# B&R Automation Studio project Parker_BMM_ST_V5_3147_V12 (part 26)

#### extruder.c - Implementation code
```c
/********************************************************************
 * COPYRIGHT --
 ********************************************************************
 * Program: extruder
 * File: extruder.c
 * Author: lij
 * Created: January 05, 2015
 ********************************************************************
 * Implementation of program extruder
 ********************************************************************/

#include <bur/plctypes.h>

#ifdef _DEFAULT_INCLUDES
	#include <AsDefault.h>
#endif

/**************************************************************************************
** 					               include user files								 **
**************************************************************************************/
#include "edge.h"               /*edge function                         */
#include "keyap2100.h"
//#include "keyap880.h"
#include "pic_id.h"

/**************************************************************************************
** 					 	                 define								                   **
**************************************************************************************/
#define     S$EXTRUDER_WAIT		           	 0
#define     S$EXTRUDER_CONTACTOR_ON		   	10
#define     S$EXTRUDER_POWER_ON_DELAY			20
#define     S$EXTRUDER_POWER_ON		        	30
#define     S$EXTRUDER_READY		       		100
#define     S$EXTRUDER_BASIC_ZONE		  		110
#define     S$EXTRUDER_PRODUCTION_ZONE	   	130
#define     S$EXTRUDER_DEC_ZONE		       	150
#define     S$EXTRUDER_POWER_OFF_DECEL			200
#define     S$EXTRUDER_POWER_OFF_PROTECT		210
#define     S$EXTRUDER_POWER_OFF_DELAY			220
/**************************************************************************************
                               Function Declarations
**************************************************************************************/
void SpeedUpDw(short ins_des,short command,speedAdjust_typ * pSpeedUpDwData);

void ExtruderCtrl(Extruder_Ctrl_typ * pExtruder,Extruder_Para_typ * pExtrPara,speedAdjust_typ * pSpeedUpDwData, Lubricate_Check_typ * pLubricCheck);

/**************************************************************************************
     	        	       I N I T U P  O F   T H E   T A S K
**************************************************************************************/
void _INIT extruderINIT(void)
{
	/* TODO: Add code here */
    RTInfo_Task.enable = 1;
    RTInfo(&RTInfo_Task);

    tTask = RTInfo_Task.cycle_time/1000.0/1000.0;		/*  from us ---> s  */

    MotorSpeedA.minVal  	  = 0;
    MotorSpeedA.frequence	  = 30;
    MotorSpeedA.waitTimeSlow = 200;
    MotorSpeedA.waitTimeFast = 500;
    MotorSpeedA.unitsSlow    = 1;
    MotorSpeedA.unitsFast	= 5;
    MotorSpeedA.unitsVFast	= 20;

    MotorSpeedA.maxVal = 100;
    MotorSpeedA.minVal = 0;

    MotorSpeedB.minVal  	 = 0;
    MotorSpeedB.frequence	 = 30;
    MotorSpeedB.waitTimeSlow = 200;
    MotorSpeedB.waitTimeFast = 500;
    MotorSpeedB.unitsSlow    = 1;
    MotorSpeedB.unitsFast	 = 5;
    MotorSpeedB.unitsVFast	 = 20;

    MotorSpeedB.maxVal = 100;
    MotorSpeedB.minVal = 0;

    MotorSpeedVisu.frequence	= 30;
    MotorSpeedVisu.waitTimeSlow = 200;
    MotorSpeedVisu.waitTimeFast = 500;
    MotorSpeedVisu.unitsSlow    = 1;
    MotorSpeedVisu.unitsFast	= 5;
    MotorSpeedVisu.unitsVFast	= 20;

    MotorSpeedVisu.maxVal = 100;
    MotorSpeedVisu.minVal = 0;

    cntExtruderStopDelay = 0;

    gExtruderA.Step = S$EXTRUDER_WAIT;
    gExtruderB.Step = S$EXTRUDER_WAIT;
    gExtruderVisu.Step = S$EXTRUDER_WAIT;

    gExtruderA.tTask  = tTask;
    gExtruderB.tTask  = tTask;
    gExtruderVisu.tTask = tTask;

	bHideCurrencyA = 0;
	bHideMeltTempA = 1;
	bHidePressureA = 1;

	bHideCurrencyB = 0;
	bHideMeltTempB = 1;
	bHidePressureB = 1;

	bHideCurrencyV = 1;
	bHideMeltTempV = 1;
	bHidePressureV = 1;

}
/**************************************************************************************
        				   C Y C L I C   P A R T   O F   T H E   T A S K
**************************************************************************************/
void _CYCLIC extruderCYCLIC(void)
{
	if(0 == gMachineFix.ExtruderA.RPM10v )gMachineFix.ExtruderA.RPM10v = 1500;
	if(0 == gMachineFix.ExtruderB.RPM10v)gMachineFix.ExtruderB.RPM10v  = 1500;
	if(0 == gMachineFix.ExtruderVisu.RPM10v )gMachineFix.ExtruderVisu.RPM10v = 1500;

	if(0 == gMachineFix.ExtruderA.Currency10V )gMachineFix.ExtruderA.Currency10V = 50;
	if(0 == gMachineFix.ExtruderB.Currency10V)gMachineFix.ExtruderB.Currency10V= 50;
	if(0 == gMachineFix.ExtruderVisu.Currency10V )gMachineFix.ExtruderVisu.Currency10V = 50;

	/*  -------------------- Extruder motor speed and current -------------------------- */
	if(gMachineOut.ExtrA_On)
	{
		gExtruderA.MotorRPM = gExtruderA.aiActRPM/32767.0  * gMachineFix.ExtruderA.RPM10v;
		gExtruderA.Current  = gExtruderA.aiCurrent/32767.0 * gMachineFix.ExtruderA.Currency10V;
		gExtruderA.ActRPM   = gExtruderA.ActSpeed/100.0  * gMachineFix.ExtruderA.RPM10v;
	}
	else
	{
		gExtruderA.MotorRPM = 0.0;
		gExtruderA.Current  = 0.0;
		gExtruderA.ActRPM   = 0.0;
	}

	if(gMachineOut.ExtrB_On)
	{
		gExtruderB.MotorRPM = gExtruderB.aiActRPM/32767.0  * gMachineFix.ExtruderB.RPM10v;
		gExtruderB.Current  = gExtruderB.aiCurrent/32767.0 * gMachineFix.ExtruderB.Currency10V;
	}
	else
	{
		gExtruderB.MotorRPM = 0.0;
		gExtruderB.Current  = 0.0;
	}

	if(gMachineOut.ExtrVisu_On)
	{
		gExtruderVisu.MotorRPM = gExtruderVisu.aiActRPM/32767.0  * gMachineFix.ExtruderVisu.RPM10v;
		gExtruderVisu.Current  = gExtruderVisu.aiCurrent/32767.0 * gMachineFix.ExtruderVisu.Currency10V;
	}
	else
	{
		gExtruderVisu.MotorRPM = 0.0;
		gExtruderVisu.Current  = 0.0;
	}

	/* ------------------ Extruder zero and max pressure ------------------ */
	if((1 == btnZeroExtrA) && (0 == btnZeroExtrA_POS))
	{
		gMachineFix.ExtruderA.MeltP0V = gExtruderA.aiMeltPressure/3276.7;
		gRecipeOperate.OnceSave = 1;
	}

	if(1 == btnMaxExtrA)
	{
		gMachineOut.MeltPrShunt = 1;
		tMaxExtrA = tMaxExtrA + tTask;
	}
	else
	{
		tMaxExtrA = 0.0;
	}

	if(tMaxExtrA > 3.0 - tTask  && tMaxExtrA < 3.0 + tTask  )
	{
		gMachineFix.ExtruderA.MeltP10V = gExtruderA.aiMeltPressure/3276.7;
		gRecipeOperate.OnceSave = 1;
	}

	if((1 == btnZeroExtrB) && (0 == btnZeroExtrB_POS))
	{
		gMachineFix.ExtruderB.MeltP0V = gHardWare.AI4632_3[1]/3276.7;		/* no this input  */
		gRecipeOperate.OnceSave = 1;
	}

	if(1 == btnMaxExtrB)
	{
		gMachineOut.MeltPrShunt = 1;
		tMaxExtrB = tMaxExtrB + tTask;
	}
	else
	{
		tMaxExtrB = 0.0;
	}

	if(tMaxExtrB > 3.0 - tTask  && tMaxExtrB < 3.0 + tTask )
	{
		gMachineFix.ExtruderB.MeltP10V = gHardWare.AI4632_3[1]/3276.7;
		gRecipeOperate.OnceSave = 1;
	}

	if(0 == btnMaxExtrA && 0 == btnMaxExtrB)
	{
		gMachineOut.MeltPrShunt = 0;
	}
	/*  -------------------- Melt pressure alarm  -------------------------- */
	if(gMachineFix.ExtruderA.WarningMeltP < 50)gMachineFix.ExtruderA.WarningMeltP = 50.0;
	if(gMachineFix.ExtruderA.AlarmMeltP < 100)gMachineFix.ExtruderA.AlarmMeltP = 100.0;

	if(gExtruderA.aiMeltPressure != 32767)
	{
		if(gExtruderA.MeltPressure > gMachineFix.ExtruderA.AlarmMeltP)
		{
			if(0 == btnMaxExtrA)
			{
				gAlarm.ExtrAMeltP_Alarm = 1;
				gAlarm.ExtrAMeltP_Warn  = 0;
			}
		}
		else if(gExtruderA.MeltPressure > gMachineFix.ExtruderA.WarningMeltP)
		{
			gAlarm.ExtrAMeltP_Alarm = 0;
			gAlarm.ExtrAMeltP_Warn  = 1;
		}
		else
		{
			gAlarm.ExtrAMeltP_Alarm = 0;
			gAlarm.ExtrAMeltP_Warn  = 0;
		}
	}
	else
	{
		gAlarm.ExtrAMeltP_Alarm = 0;
		gAlarm.ExtrAMeltP_Warn  = 0;
	}

	/* --------------------  current alarm and warning -------------------- */
	if(gMachineFix.ExtruderA.WarningCurrent < 2)gMachineFix.ExtruderA.WarningCurrent = 2;
	if(gMachineFix.ExtruderA.AlarmCurrent   < 5)gMachineFix.ExtruderA.AlarmCurrent = 5;

	if(gExtruderA.aiCurrent != 32767)
	{
		if(gExtruderA.Current > gMachineFix.ExtruderA.AlarmCurrent)
		{
			tAlarmCurentA = tAlarmCurentA+tTask;
			if(tAlarmCurentA > 10000)tAlarmCurentA= 1000;
			tWarnCurentA  = 0.0;
		}
		else if(gExtruderA.Current > gMachineFix.ExtruderA.WarningCurrent)
		{
			tAlarmCurentA = 0.0;
			tWarnCurentA = tWarnCurentA+tTask;
			if(tWarnCurentA > 10000)tWarnCurentA = 1000;
		}
		else
		{
			tWarnCurentA = 0.0;
			tAlarmCurentA = 0.0;
		}

		if(tAlarmCurentA > 5.0)
		{
			gAlarm.ExtrACurrentAlarm = 1;
		}
		else
		{
			gAlarm.ExtrACurrentAlarm = 0;
		}

		if(tWarnCurentA > 5.0)
		{
			gAlarm.ExtrACurrentWarn = 1;
		}
		else
		{
			gAlarm.ExtrACurrentWarn = 0;
		}
	}
	else
	{
		tWarnCurentA = 0.0;
		tAlarmCurentA = 0.0;

		gAlarm.ExtrACurrentWarn = 0;
		gAlarm.ExtrACurrentAlarm = 0;
	}

	if(gMachineFix.ExtruderB.WarningCurrent < 2)gMachineFix.ExtruderB.WarningCurrent = 2;
	if(gMachineFix.ExtruderB.AlarmCurrent   < 5)gMachineFix.ExtruderB.AlarmCurrent = 5;

	if(gExtruderB.aiCurrent != 32767)
	{
		if(gExtruderB.Current > gMachineFix.ExtruderB.AlarmCurrent)
		{
			tAlarmCurentB = tAlarmCurentB+tTask;
			if(tAlarmCurentB > 10000)tAlarmCurentB= 1000;
			tWarnCurentB  = 0.0;
		}
		else if(gExtruderB.Current > gMachineFix.ExtruderB.WarningCurrent)
		{
			tAlarmCurentB = 0.0;
			tWarnCurentB = tWarnCurentB+tTask;
			if(tWarnCurentB > 10000)tWarnCurentB = 1000;
		}
		else
		{
			tWarnCurentB = 0.0;
			tAlarmCurentB = 0.0;
		}

		if(tAlarmCurentB > 5.0)
		{
			gAlarm.ExtrBCurrentAlarm = 1;
		}
		else
		{
			gAlarm.ExtrBCurrentAlarm = 0;
		}

		if(tWarnCurentB > 5.0)
		{
			gAlarm.ExtrBCurrentWarn = 1;
		}
		else
		{
			gAlarm.ExtrBCurrentWarn = 0;
		}
	}
	else
	{
		tWarnCurentB = 0.0;
		tAlarmCurentB = 0.0;

		gAlarm.ExtrBCurrentWarn = 0;
		gAlarm.ExtrBCurrentAlarm = 0;
	}

	/* -------------------- Hopper cooling  -------------------------- */
	bHideHopperCooling = !gMachineFix.Option.bHopperCooling;
	gMachineFix.Option.bHopperCooling =0; //ipis0319
	if(1 == gMachineFix.Option.bHopperCooling)
	{
		if(!gMachinePara.HopperCoolStart)gMachinePara.HopperCoolStart = 65;
		if(!gMachinePara.HopperCoolStop )gMachinePara.HopperCoolStop = 55;

		if(gMachineInfo.TempHopper > gMachinePara.HopperCoolStart)
		{
			gMachineOut.HopperCoolingA = 1;
		}

		if(gMachineInfo.TempHopper < gMachinePara.HopperCoolStop)
		{
			gMachineOut.HopperCoolingA = 0;
		}
	}
	else
	{
		gMachineOut.HopperCoolingA = 0;
	}
	/* -------------------- Extruder motor cooling  -------------------------- */
	bHideExtrMotorCooling = !gMachineFix.Option.bExtruderMotorCooling;
	gMachineFix.Option.bExtruderMotorCooling=0; //ipis0319
	if(!gMachinePara.ExtruderA.TempCoolStart)gMachinePara.ExtruderA.TempCoolStart = 75;
	if(!gMachinePara.ExtruderA.TempCoolStop)gMachinePara.ExtruderA.TempCoolStop = 65;
	if(!gMachinePara.ExtrLiftLower.warningMotorTemp)gMachinePara.ExtrLiftLower.warningMotorTemp= 90;
	if(!gMachinePara.ExtrLiftLower.AlarmMotorTemp)gMachinePara.ExtrLiftLower.AlarmMotorTemp = 100;

	if(1 == gMachineFix.Option.bExtruderMotorCooling)
	{
		if(gMachineInfo.TempExtrCoolWater > gMachinePara.ExtruderA.TempCoolStart)
		{
			gMachineOut.ExtrA_CoolWaterOn = 1;
		}

		if(gMachineInfo.TempExtrCoolWater < gMachinePara.ExtruderA.TempCoolStop)
		{
			gMachineOut.ExtrA_CoolWaterOn = 0;
		}

		if(gMachineInfo.TempExtrCoolWater > gMachinePara.ExtrLiftLower.warningMotorTemp)
		{
			tAlarmExtrTempA = tAlarmExtrTempA + tTask;

			if(tAlarmExtrTempA > 10000.0)tAlarmExtrTempA = 100.0;
		}
		else
		{
			tAlarmExtrTempA = 0.0;
		}

		if(tAlarmExtrTempA > 10.0)
		{
			gAlarm.A_ExtrMotorTempAlarm = 1;
		}

		if(gMachineInfo.TempExtrCoolWater > gMachinePara.ExtrLiftLower.AlarmMotorTemp)
		{
			tStopExtrTempA = tStopExtrTempA + tTask;

			if(tStopExtrTempA > 10000.0)tStopExtrTempA = 100.0;
		}
		else
		{
			tStopExtrTempA = 0.0;
		}

		if(tStopExtrTempA > 10.0)
		{
			gAlarm.A_ExtrMotorTempStop = 1;
		}

		if(0 == gMachineIn.ExtrA_ColiTempNormal)
		{
			tColiTempNormalA = tColiTempNormalA + tTask;

			if(tColiTempNormalA > 10000.0)tColiTempNormalA = 100.0;
		}
		else
		{
			tColiTempNormalA = 0.0;
		}

		if(tColiTempNormalA > 10.0)
		{
			gAlarm.A_ColiTempNormal = 1;
		}
	}
	else
	{
		gAlarm.A_ExtrMotorTempStop = 0;
		gAlarm.A_ColiTempNormal = 0;
		gMachineOut.ExtrA_CoolWaterOn = 0;
	}

   /* ----------------------- extruder key ------------------------- */
   if(1 == gMachineIn.MainControl && gPanelObj.GetPicture != PIC_INIT && gPanelObj.GetPicture != PIC_SCREEN_SAVE)
   {
     gExtruderA.bKeyOnOff       = gPanelObj.KeyMatric[S$KEYMATRIX_EXTRUDER_A];
     gExtruderB.bKeyOnOff    = gPanelObj.KeyMatric[S$KEYMATRIX_EXTRUDER_B];
	  gMachineIn.ExtrA_HopperKey = gPanelObj.KeyMatric[S$KEYMATRIX_HOPPER_A];
   }/*if(1 == gMachineIn.MainControl ..... */

   /* ----- A extruder increase or decrease speed ----- */
   if(16384 == gExtruderA.FoucsBasic || 16384 == gExtruderA.FocusProduct || PIC_SPEED != gPanelObj.GetPicture)
   {
      gExtruderA.bKeyInc = gPanelObj.KeyMatric[S$KEYMATRIX_SPEED_UP];
      gExtruderA.bKeyDec = gPanelObj.KeyMatric[S$KEYMATRIX_SPEED_DN];
   }
   else
   {
      gExtruderA.bKeyInc = 0;
      gExtruderA.bKeyDec = 0;
   }
   gExtruderA.tProtect = gMachineFix.ExtruderA.tProtect;
   gExtruderA.tOnDelay = gMachineFix.ExtruderA.tOnDelay;
   gExtruderA.tOffDelay = gMachineFix.ExtruderA.tOffDelay;

	LubricCheckA.diLubricCheck = gMachineIn.ExtrA_LubrNormal;
	LubricCheckA.tSetCheckTime = gMachineFix.ExtruderA.tLubricateCheck;

   ExtruderCtrl(&gExtruderA, &gMachinePara.ExtruderA, &MotorSpeedA, &LubricCheckA);
   gMachineOut.ExtrA_On = gExtruderA.doOn;

	gAlarm.A_ExtrLubricCheck = LubricCheckA.bLubricError;
//	gAlarm.A_ExtruderMotorOverload = gMachineIn.ExtrA_MotorErr;

	/* extruder A on and feedback  */
	gMachineIn.ExtrA_OnOff = gMachineOut.ExtrA_On;
	if(gMachineOut.ExtrA_On != gMachineIn.ExtrA_OnOff)
	{
		tExtrA_OnNormal = tExtrA_OnNormal + tTask;
		if(tExtrA_OnNormal >= 600.0)tExtrA_OnNormal = 60.0;
	}
	else
	{
		tExtrA_OnNormal = 0.0;
	}

	if(tExtrA_OnNormal >= 30.0)
	{
		gExtruderA.OnFeedbackErr = 1;
		gAlarm.ExtrA_NotOn = 1;
	}
	else
	{
		gExtruderA.OnFeedbackErr = 0;
	}

	/*  extruder A hopper  */
	if(1 == gMachineIn.ExtrA_HopperKey && 0 == ExtrA_HopperKeyOld)
	{
		if((1 == gMachineIn.ExtrA_OnOff) && (gExtruderA.Out > 0.0))
		{
			gMachineOut.HopperGateOpenA = !gMachineOut.HopperGateOpenA;
		}
		else
		{
			if(0 == gMachineIn.ExtrA_OnOff)gImply.ExtruderA_NotOn = 1;
			if(0.0 == gExtruderA.Out)gImply.ExtruderA_NotOut = 1;
		}
	}
	ExtrA_HopperKeyOld = gMachineIn.ExtrA_HopperKey;

	if((0 == gMachineIn.ExtrA_OnOff) || (0.0 == gExtruderA.Out))
	{
		if(1 == gMachineOut.HopperGateOpenA)
		{
			if(0 == gMachineIn.ExtrA_OnOff)gImply.ExtruderA_NotOn = 1;
			if(0.0 == gExtruderA.Out)gImply.ExtruderA_NotOut = 1;
			gMachineOut.HopperGateOpenA = 0;
		}
	}

   /* ----- B extruder increase or decrease speed ----- */
   if(16384 == gExtruderB.FoucsBasic || 16384 == gExtruderB.FocusProduct)
   {
      gExtruderB.bKeyInc = gPanelObj.KeyMatric[S$KEYMATRIX_SPEED_UP];
      gExtruderB.bKeyDec = gPanelObj.KeyMatric[S$KEYMATRIX_SPEED_DN];
   }
   else
   {
      gExtruderB.bKeyInc = 0;
      gExtruderB.bKeyDec = 0;
   }
   gExtruderB.tProtect = gMachineFix.ExtruderA.tProtect;
   gExtruderB.tOnDelay = gMachineFix.ExtruderA.tOnDelay;
   gExtruderB.tOffDelay = gMachineFix.ExtruderA.tOffDelay;

	LubricCheckB.diLubricCheck = gMachineIn.ExtrB_LubrNormal;
	LubricCheckB.tSetCheckTime = gMachineFix.ExtruderA.tLubricateCheck;

   ExtruderCtrl(&gExtruderB, &gMachinePara.ExtruderB, &MotorSpeedB, &LubricCheckB);
   gMachineOut.ExtrB_On = gExtruderB.doOn;

	gAlarm.B_ExtrLubricCheck = LubricCheckB.bLubricError;
//	gAlarm.B_ExtruderMotorOverload = gMachineIn.ExtrB_MotorErr;

	/* extruder B on and feedback  */
	gMachineIn.ExtrB_OnOff = gMachineOut.ExtrB_On;
	if(gMachineOut.ExtrB_On != gMachineIn.ExtrB_OnOff)
	{
		tExtrB_OnNormal = tExtrA_OnNormal + tTask;
		if(tExtrB_OnNormal >= 600.0)tExtrB_OnNormal = 60.0;
	}
	else
	{
		tExtrB_OnNormal = 0.0;
	}

	if(tExtrB_OnNormal >= 30.0)
	{
		gExtruderB.OnFeedbackErr = 1;
		gAlarm.ExtrB_NotOn = 1;
	}
	else
	{
		gExtruderB.OnFeedbackErr = 0;
	}

	if(1 == gMachineIn.ExtrB_HopperKey && 0 == ExtrB_HopperKeyOld)
	{
		if((1 == gMachineIn.ExtrB_OnOff) && (gExtruderB.Out > 0.0))
		{
			gMachineOut.HopperGateOpenB = !gMachineOut.HopperGateOpenB;
		}
		else
		{
			if(0 == gMachineIn.ExtrB_OnOff)gImply.ExtruderB_NotOn = 1;
			if(0.0 == gExtruderB.Out)gImply.ExtruderB_NotOut = 1;
		}
	}
	ExtrB_HopperKeyOld = gMachineIn.ExtrB_HopperKey;

	if((0 == gMachineIn.ExtrB_OnOff) || (0.0 == gExtruderB.Out))
	{
		if(1 == gMachineOut.HopperGateOpenB)
		{
			if(0 == gMachineIn.ExtrB_OnOff)gImply.ExtruderB_NotOn = 1;
			if(0.0 == gExtruderB.Out)gImply.ExtruderB_NotOut = 1;
			gMachineOut.HopperGateOpenB = 0;
		}
	}

   /* ----- Visual extruder increase or decrease speed ----- */
   if(16384 == gExtruderVisu.FoucsBasic || 16384 == gExtruderVisu.FocusProduct)
   {
      gExtruderVisu.bKeyInc = gPanelObj.KeyMatric[S$KEYMATRIX_SPEED_UP];
      gExtruderVisu.bKeyDec = gPanelObj.KeyMatric[S$KEYMATRIX_SPEED_DN];
   }
   else
   {
      gExtruderVisu.bKeyInc = 0;
      gExtruderVisu.bKeyDec = 0;
   }
   gExtruderVisu.tProtect = gMachineFix.ExtruderA.tProtect;
   gExtruderVisu.tOnDelay = gMachineFix.ExtruderA.tOnDelay;
   gExtruderVisu.tOffDelay = gMachineFix.ExtruderA.tOffDelay;

	LubricCheckVisu.diLubricCheck = 1;
	LubricCheckVisu.tSetCheckTime = gMachineFix.ExtruderA.tLubricateCheck;

   ExtruderCtrl(&gExtruderVisu, &gMachinePara.ExtruderVisu, &MotorSpeedVisu, &LubricCheckVisu);
   gMachineOut.ExtrVisu_On = gExtruderVisu.doOn;

	gAlarm.VisuExtrMotorOverload = gMachineIn.ExtrV_MotorErr;
	gAlarm.VisuExtrCoolOverload  = gMachineIn.ExtrV_CoolMotorErr;

	/* extruder A on and feedback  */
	if(gMachineOut.ExtrVisu_On != gMachineIn.ExtrV_OnOff)
	{
		tExtrV_OnNormal = tExtrV_OnNormal + tTask;
		if(tExtrV_OnNormal >= 600.0)tExtrV_OnNormal = 60.0;
	}
	else
	{
		tExtrV_OnNormal = 0.0;
	}

	if(tExtrV_OnNormal >= 30.0)
	{
		gExtruderVisu.OnFeedbackErr = 1;
		gAlarm.ExtrV_NotOn = 1;
	}
	else
	{
		gExtruderVisu.OnFeedbackErr = 0;
	}

   gMachineInfo.Extruder       = gMachineOut.ExtrA_On;
   gMachineOut.ExtruderCooling = gMachineInfo.Extruder;

   /* ----------------------- Stop extruder ----------------------- */
   /* ----- A extruder ----- */
   gExtruderA.bKeyOff = 0;
   if (1 == gMachineInfo.ExtrTLow     || 0 == gMachineInfo.IsHeat           || 0 == gMachineIn.ParisonPumpRunning   ||
       1 == gMachineIn.ExtrA_MotorErr || 1 == gMachineIn.ExtrA_CoolMotorErr || 1 == gAlarm.A_ExtrMotorTempStop      ||
		 1 == gAlarm.ExtrACurrentAlarm)
   {
		if(1 == gMachineOut.ExtrA_On)
		{
			if(1 == gMachineInfo.ExtrTLow)gAlarm.ScrewTempLow = 1;
			if(0 == gMachineInfo.IsHeat)gAlarm.HeatingNotOn = 1;
			if(0 == gMachineIn.ParisonPumpRunning)gAlarm.ParisonPumpNotOn = 1;
//			gAlarm.A_ExtruderMotorOverload = gMachineIn.ExtrA_MotorErr;
			gExtruderA.bKeyOff = 1;
		}
   }

   /* ----- B extruder ----- */
   gExtruderB.bKeyOff = 0;
   if (1 == gMachineInfo.ExtrTLow     || 0 == gMachineInfo.IsHeat           || 0 == gMachineIn.ParisonPumpRunning ||
       1 == gMachineIn.ExtrB_MotorErr || 1 == gMachineIn.ExtrB_CoolMotorErr || 1 == gAlarm.ExtrBCurrentAlarm)
   {
		if(1 == gMachineOut.ExtrB_On)
		{
			if(1 == gMachineInfo.ExtrTLow)gAlarm.ScrewTempLow = 1;
			if(0 == gMachineInfo.IsHeat)gAlarm.HeatingNotOn = 1;
			if(0 == gMachineIn.ParisonPumpRunning)gAlarm.ParisonPumpNotOn = 1;
//			gAlarm.B_ExtruderMotorOverload = gMachineIn.ExtrB_MotorErr;
			gExtruderB.bKeyOff = 1;
		}
   }

   /* ----- Visual extruder ----- */
   gExtruderVisu.bKeyOff = 0;
   if (1 == gMachineInfo.ExtrTLow     || 0 == gMachineInfo.IsHeat || 0 == gMachineIn.ParisonPumpRunning ||
       1 == gMachineIn.ExtrV_MotorErr || 1 == gMachineIn.ExtrV_CoolMotorErr || 0 == gMachineIn.ExtrA_OnOff)
   {
		if(1 == gMachineOut.ExtrVisu_On)
		{
			if(1 == gMachineInfo.ExtrTLow)gAlarm.ScrewTempLow = 1;
			if(0 == gMachineInfo.IsHeat)gAlarm.HeatingNotOn = 1;
			if(0 == gMachineIn.ParisonPumpRunning)gAlarm.ParisonPumpNotOn = 1;
			gAlarm.VisuExtrMotorOverload = gMachineIn.ExtrV_MotorErr;
			if(0 == gMachineIn.ExtrA_OnOff)gAlarm.ExtrA_NotOn = 1;
			gExtruderVisu.bKeyOff = 1;
		}
   }

   /* ------------------------ Auto error stop extruder ---------------------------- */
   if(1 == gPROCESS_info.extruderStopEnable)
   {
     cntExtruderStopDelay ++;
   }
   else
   {
     cntExtruderStopDelay = 0;
   }

   if(gMachineFix.ExtruderA.StopTime <= 0.0)gMachineFix.ExtruderA.StopTime = 3.0;
   if(gMachineFix.ExtruderA.StopTime < cntExtruderStopDelay * tTask)
   {
     if(1 == gTKmanual.Status)
     {
         gExtruderA.bKeyOff = 1;
         gExtruderB.bKeyOff = 1;
		 gExtruderD.bKeyOff = 1;
         gExtruderVisu.bKeyOff = 1;
         gPROCESS_info.extruderStopEnable = 0;
         cntExtruderStopDelay = 0;
     }
   }
}
/**************************************************************************************
        				   E X I T   P A R T   O F   T H E   T A S K
**************************************************************************************/
void _EXIT extruderEXIT(void)
{
	/* TODO: Add code here */
}

/* adjust the speed of motor*/
void SpeedUpDw(short ins_des,short command,speedAdjust_typ * pSpeedUpDwData)
{
    unsigned short index;

    if(pSpeedUpDwData->pSpeed != 0)  /*  point is not NULL  */
    {
        index = ins_des + 1;

        if (command == 1)
        {
            pSpeedUpDwData->iSpeed[index]++;
            pSpeedUpDwData->iSpeed[index+1]++;
            if (pSpeedUpDwData->iSpeed[index+1] == 1) (*pSpeedUpDwData->pSpeed) = (*pSpeedUpDwData->pSpeed) + pSpeedUpDwData->unitsSlow*ins_des;
            if (pSpeedUpDwData->iSpeed[index]>pSpeedUpDwData->frequence) pSpeedUpDwData->iSpeed[index] = 0;

            if (pSpeedUpDwData->iSpeed[index+1]<50) ;
            else if (pSpeedUpDwData->iSpeed[index+1]<pSpeedUpDwData->waitTimeSlow)
            {
                if (pSpeedUpDwData->iSpeed[index]== 0) (*pSpeedUpDwData->pSpeed) = (*pSpeedUpDwData->pSpeed) + pSpeedUpDwData->unitsSlow*ins_des;
            }
            else if (pSpeedUpDwData->iSpeed[index+1]<pSpeedUpDwData->waitTimeFast)
            {
                if (pSpeedUpDwData->iSpeed[index] == 0) (*pSpeedUpDwData->pSpeed) = (*pSpeedUpDwData->pSpeed) + pSpeedUpDwData->unitsFast*ins_des;
            }
            else
            {
                if (pSpeedUpDwData->iSpeed[index] == 0) (*pSpeedUpDwData->pSpeed) = (*pSpeedUpDwData->pSpeed) + pSpeedUpDwData->unitsVFast*ins_des;
                pSpeedUpDwData->iSpeed[index+1] = pSpeedUpDwData->waitTimeFast;
            }
        }
        else
        {
            pSpeedUpDwData->iSpeed[index] = 0;
            pSpeedUpDwData->iSpeed[index+1] = 0;
        }
        if ((*pSpeedUpDwData->pSpeed) >= pSpeedUpDwData->maxVal) (*pSpeedUpDwData->pSpeed) = pSpeedUpDwData->maxVal;
        if ((*pSpeedUpDwData->pSpeed) <= pSpeedUpDwData->minVal) (*pSpeedUpDwData->pSpeed) = pSpeedUpDwData->minVal;
    }/*  if(pSpeedUpDwData->pSpeed != 0) */
}/*end of function*/

/* ---------- Extruder contorl ---------- */
void ExtruderCtrl(Extruder_Ctrl_typ * pExtruder, Extruder_Para_typ * pExtrPara, speedAdjust_typ * pSpeedUpDwData, Lubricate_Check_typ * pLubricCheck)
{
    if(pExtruder->tOnDelay  < pExtruder->tTask * 2.0)pExtruder->tOnDelay = pExtruder->tTask * 2.0;
    if(pExtruder->tOffDelay < pExtruder->tTask * 2.0)pExtruder->tOffDelay= pExtruder->tTask * 2.0;

    if(pExtruder->tTask <= 0.0)
    {
        pExtruder->tET_s = 0.0;
        pExtruder->LedOn = 0;
        pExtruder->LedProduction = 0;

        pExtruder->doContactor = 0;
        pExtruder->doOn = 0;
        pExtruder->Out = 0.0;

        pExtruder->bKeyOnOff = 0;
        pExtruder->bKeyOff = 0;
        pExtruder->bKeyOnOffOld = 0;
        pExtruder->bKeyOffOld = 0;

        pExtruder->Step = S$EXTRUDER_WAIT;
        return;
    }

    /*  On Off button edge start */
    if(1 == pExtruder->bKeyOnOff && 0 == pExtruder->bKeyOnOffOld)
    {
        if(S$EXTRUDER_WAIT == pExtruder->Step)
        {
				pExtruder->LedOn = 1;
            pExtruder->Step = S$EXTRUDER_CONTACTOR_ON;
        }
        else
        {
				pExtruder->LedOn = 0;
            if(pExtruder->Step < S$EXTRUDER_POWER_ON && pExtruder->Step > S$EXTRUDER_WAIT)
            {
               pExtruder->Step = S$EXTRUDER_WAIT;
            }
            else if(pExtruder->Step >= S$EXTRUDER_POWER_ON && pExtruder->Step < S$EXTRUDER_POWER_OFF_DECEL)
            {
                if(pExtruder->Step > S$EXTRUDER_BASIC_ZONE)
                {
                    pExtruder->Step = S$EXTRUDER_POWER_OFF_DECEL;
                }
                else
                {
                    pExtruder->Step = S$EXTRUDER_POWER_OFF_PROTECT;
                }
            }
        }
    }
    pExtruder->bKeyOnOffOld = pExtruder->bKeyOnOff;

    /* -------- internal stop -------- */
    if(1 == pExtruder->bKeyOff)
    {
		 pExtruder->LedOn = 0;
       if(pExtruder->Step < S$EXTRUDER_POWER_ON && pExtruder->Step > S$EXTRUDER_WAIT)
       {
          pExtruder->Step = S$EXTRUDER_WAIT;
       }
       else if(pExtruder->Step >= S$EXTRUDER_POWER_ON && pExtruder->Step < S$EXTRUDER_POWER_OFF_DECEL)
       {
          if(pExtruder->Step > S$EXTRUDER_BASIC_ZONE)
          {
             pExtruder->Step = S$EXTRUDER_POWER_OFF_DECEL;
          }
          else
          {
             pExtruder->Step = S$EXTRUDER_POWER_OFF_PROTECT;
          }
       }
    }
    pExtruder->bKeyOffOld = pExtruder->bKeyOff;

	if(1 == pExtruder->bKeyStop)
	{
		pExtruder->bKeyStop = 0;
		if(pExtruder->Step < S$EXTRUDER_POWER_ON && pExtruder->Step > S$EXTRUDER_WAIT)
		{
			pExtruder->Step = S$EXTRUDER_WAIT;
		}
		else if(pExtruder->Step >= S$EXTRUDER_POWER_ON && pExtruder->Step < S$EXTRUDER_POWER_OFF_DECEL)
		{
			if(pExtruder->Step > S$EXTRUDER_BASIC_ZONE)
			{
				pExtruder->Step = S$EXTRUDER_POWER_OFF_DECEL;
			}
			else
			{
				pExtruder->Step = S$EXTRUDER_POWER_OFF_PROTECT;
			}
		}
	}

    /*  ------ motor protection ------- */
    if(pExtruder->doOnOld != pExtruder->doOn && pExtruder->tTask > 0.0)
    {
        pExtruder->cntProtect = pExtruder->tProtect /pExtruder->tTask;
    }

    if(pExtruder->cntProtect > 0)pExtruder->cntProtect--;

    /* ----- step machine control ----- */
    switch(pExtruder->Step)
    {
        case S$EXTRUDER_WAIT:
            pExtruder->tET_s = 0.0;
            pExtruder->LedBaisic = 0;
            pExtruder->LedProduction = 0;

            pExtruder->doContactor = 0;
            pExtruder->doOn = 0;
            pExtruder->doFeedingCylFw = pExtruder->bKeyFeedingCylFw; /* manual test */
            pExtruder->Out = 0.0;
				pLubricCheck->bEnable = 0;
            break;

        case S$EXTRUDER_CONTACTOR_ON:
            pExtruder->tET_s = 0.0;
            pExtruder->LedBaisic = 0;
            pExtruder->LedProduction = 0;

            pExtruder->doContactor = 1;
            pExtruder->doFeedingCylFw = 0;
            pExtruder->Out = 0.0;
            pExtruder->Step = S$EXTRUDER_POWER_ON_DELAY;
            break;

        case S$EXTRUDER_POWER_ON_DELAY:
            pExtruder->LedBaisic = 0;
            pExtruder->LedProduction = 0;

            pExtruder->doContactor = 1;
            pExtruder->doOn = 0;
            pExtruder->doFeedingCylFw = 0;
            pExtruder->Out = 0.0;
            pExtruder->tET_s = pExtruder->tET_s + pExtruder->tTask;
            if(pExtruder->tET_s >= pExtruder->tOnDelay)
            {
                pExtruder->tET_s = 0.0;
                pExtruder->Step = S$EXTRUDER_POWER_ON;
            }
            break;

        case S$EXTRUDER_POWER_ON:
            pExtruder->tET_s = 0.0;
            pExtruder->LedBaisic = 0;
            pExtruder->LedProduction = 0;

            pExtruder->doContactor = 1;
            pExtruder->doOn = 1;
            pExtruder->Out = 0.0;
            pExtruder->doFeedingCylFw = 0;

            pExtruder->Step = S$EXTRUDER_READY;
            break;

        case S$EXTRUDER_READY:
            pExtruder->tET_s = 0.0;
            pExtruder->LedBaisic = 0;
            pExtruder->LedProduction = 0;

            pExtruder->doContactor = 1;
            pExtruder->doOn = 1;
            pExtruder->doFeedingCylFw = 0;
            pExtruder->Out = 0.0;

				pLubricCheck->bEnable = 1;
				pLubricCheck->bLubricError = 0;

            if(1 == EDGEPOS(pExtruder->bKeyBasic,pExtruder->bKeyBasicOld))
            {
                pExtruder->Step = S$EXTRUDER_BASIC_ZONE;
            }
            break;

        case S$EXTRUDER_BASIC_ZONE:
            pExtruder->tET_s = 0.0;
            pExtruder->LedBaisic = 1;
            pExtruder->LedProduction = 0;

            pSpeedUpDwData->maxVal = 50;

				pSpeedUpDwData->pSpeed = &pExtrPara->BasicSpeed;
            SpeedUpDw(1   , pExtruder->bKeyInc , pSpeedUpDwData);
            SpeedUpDw(- 1 , pExtruder->bKeyDec , pSpeedUpDwData);
				pExtruder->BasicSpeed = pExtrPara->BasicSpeed;

            pExtruder->doContactor = 1;
            pExtruder->doOn = 1;
            pExtruder->doFeedingCylFw = 0;
            pExtruder->Out = pExtruder->BasicSpeed;

            if(1 == EDGEPOS(pExtruder->bKeyProduction,pExtruder->bKeyProductionOld))
            {
                pExtruder->Step = S$EXTRUDER_PRODUCTION_ZONE;
            }
            break;

        case S$EXTRUDER_PRODUCTION_ZONE:
            pExtruder->tET_s = 0.0;
            pExtruder->LedBaisic = 0;
            pExtruder->LedProduction = 1;

            pSpeedUpDwData->maxVal = 100;

				pSpeedUpDwData->pSpeed = &pExtrPara->ProductionSpeed;
            SpeedUpDw(1   , pExtruder->bKeyInc , pSpeedUpDwData);
            SpeedUpDw(- 1 , pExtruder->bKeyDec , pSpeedUpDwData);
				pExtruder->ProductionSpeed = pExtrPara->ProductionSpeed;

            pExtruder->doContactor = 1;
            pExtruder->doOn = 1;
            pExtruder->doFeedingCylFw = 1;
            pExtruder->Out = pExtruder->ProductionSpeed;

            if(1 == EDGEPOS(pExtruder->bKeyBasic,pExtruder->bKeyBasicOld))
            {
                pExtruder->Step = S$EXTRUDER_BASIC_ZONE;
            }
            break;

        case S$EXTRUDER_DEC_ZONE:
            pExtruder->tET_s = 0.0;
            pExtruder->LedBaisic = 0;
            pExtruder->LedProduction = 0;

            pExtruder->doContactor = 1;
            pExtruder->doOn = 1;
            pExtruder->doFeedingCylFw = 1;
            pExtruder->Out = pExtruder->BasicSpeed;

            if(pExtruder->ActSpeed <= pExtruder->BasicSpeed + 0.01)
            {
                pExtruder->Step = S$EXTRUDER_READY;
            }
            break;

        /* power off step  */
        case S$EXTRUDER_POWER_OFF_DECEL:
            pExtruder->tET_s = 0.0;
            pExtruder->LedBaisic = 0;
            pExtruder->LedProduction = 0;

            pExtruder->doContactor = 1;
            pExtruder->doOn = 1;
            pExtruder->doFeedingCylFw = 0;
            pExtruder->Out = pExtruder->BasicSpeed;

            if(pExtruder->ActSpeed <= pExtruder->BasicSpeed + 0.01)
            {
                pExtruder->Step = S$EXTRUDER_POWER_OFF_PROTECT;
            }
            break;

        case S$EXTRUDER_POWER_OFF_PROTECT:
            pExtruder->tET_s = 0.0;
            pExtruder->LedBaisic = 0;
            pExtruder->LedProduction = 0;

            pExtruder->doContactor = 1;
            pExtruder->doOn = 1;
            pExtruder->doFeedingCylFw = 0;
            pExtruder->Out = 0.0;

            if(0 == pExtruder->cntProtect)
            {
                pExtruder->Step = S$EXTRUDER_POWER_OFF_DELAY;
            }
            break;

        case S$EXTRUDER_POWER_OFF_DELAY:
            pExtruder->LedBaisic = 0;
            pExtruder->LedProduction = 0;

            pExtruder->doContactor = 1;
            pExtruder->doFeedingCylFw = 0;
            pExtruder->Out = 0.0;
            pExtruder->tET_s = pExtruder->tET_s + pExtruder->tTask;
            if(pExtruder->tET_s >= pExtruder->tOffDelay)
            {
	            pExtruder->tET_s = 0.0;
					if(0 == pExtruder->LedOn)
					{
						pExtruder->Step = S$EXTRUDER_WAIT;
					}
					else
					{
						pExtruder->Step = S$EXTRUDER_READY;
					}
            }
            break;
    }/* switch( pExtruder->Step) */

	 if(pLubricCheck->tSetCheckTime < 1.0)pLubricCheck->tSetCheckTime = 1.0;

	 if(1 == pLubricCheck->bEnable && (pExtruder->Step > S$EXTRUDER_READY && pExtruder->Step <S$EXTRUDER_DEC_ZONE))
	 {
		if(0 == pLubricCheck->diLubricCheck)
		{
			pLubricCheck->tActCheckTime = pLubricCheck->tActCheckTime + pExtruder->tTask;
			if(pLubricCheck->tActCheckTime >= pLubricCheck->tSetCheckTime * 10.0)pLubricCheck->tActCheckTime=  2.0 * pLubricCheck->tSetCheckTime;
			if(pLubricCheck->tActCheckTime >= pLubricCheck->tSetCheckTime)
			{
				pLubricCheck->bLubricError = 1;
				/*pLubricCheck->bEnable = 0;*/
			}
			else
			{
				pLubricCheck->bLubricError = 0;
			}

			pLubricCheck->tCheckDly = 5.0;
		}
		else
		{
			pLubricCheck->bLubricError = 0;
			pLubricCheck->tActCheckTime = 0.0;
		}
	 }
	 else
	 {
		pLubricCheck->tActCheckTime = 0.0;
		if(pLubricCheck->tCheckDly > 0.0)pLubricCheck->tCheckDly= pLubricCheck->tCheckDly - pExtruder->tTask;
		if(pLubricCheck->tCheckDly < 0.0)pLubricCheck->tCheckDly= 0.0;
		if(0.0 == pLubricCheck->tCheckDly)pLubricCheck->bLubricError = 0;
	 }

    pExtruder->doOnOld = pExtruder->doOn;
    pExtruder->bKeyBasicOld = pExtruder->bKeyBasic;
    pExtruder->bKeyProductionOld = pExtruder->bKeyProduction;
    pExtruder->bKeyFeedingCylFwOld = pExtruder->bKeyFeedingCylFw;
}/*end of function*/
```

#### extruder.typ - Local data types
```iecst
(********************************************************************
 * COPYRIGHT --
 ********************************************************************
 * Program: extruder
 * File: extruder.typ
 * Author: lij
 * Created: January 05, 2015
 ********************************************************************
 * Local data types of program extruder
 ********************************************************************)

TYPE
	Lubricate_Check_typ : 	STRUCT
		bEnable : BOOL;
		diLubricCheck : BOOL;
		tSetCheckTime : REAL;
		tActCheckTime : REAL;
		tCheckDly : REAL;
		bLubricError : BOOL;
	END_STRUCT;
	speedAdjust_typ : 	STRUCT
		pSpeed : REFERENCE TO REAL;
		maxVal : UINT;
		minVal : UINT;
		frequence : UINT;
		waitTimeSlow : UINT;
		waitTimeFast : UINT;
		unitsSlow : UINT;
		unitsFast : UINT;
		unitsVFast : UINT;
		iSpeed : ARRAY[0..3]OF UINT;
	END_STRUCT;
END_TYPE
```

#### extruder.var - Local variables
```iecst
(********************************************************************
 * COPYRIGHT --
 ********************************************************************
 * Program: extruder
 * File: extruder.var
 * Author: lij
 * Created: January 05, 2015
 ********************************************************************
 * Local variables of program extruder
 ********************************************************************)
VAR
	tTask : REAL := 0.0;
	RTInfo_Task : RTInfo := (0);
	tAlarmCurentA : REAL;
	tWarnCurentA : REAL;
	tAlarmCurentB : REAL;
	tWarnCurentB : REAL;
	tAlarmExtrTempA : REAL;
	tStopExtrTempA : REAL;
	tColiTempNormalA : REAL;
	bHideCurrencyA : UINT;
	bHideMeltTempA : UINT;
	bHidePressureA : UINT;
	bHideCurrencyB : UINT;
	bHideMeltTempB : UINT;
	bHidePressureB : UINT;
	bHideCurrencyV : UINT;
	bHideMeltTempV : UINT;
	bHidePressureV : UINT;
	bHideExtrMotorCooling : UINT;
	bHideHopperCooling : UINT;
	btnZeroExtrA : USINT;
	btnMaxExtrA : USINT;
	tMaxExtrA : REAL;
	btnZeroExtrB : USINT;
	btnMaxExtrB : USINT;
	tMaxExtrB : REAL;
	btnZeroExtrA_POS : USINT;
	btnZeroExtrB_POS : USINT;
	ExtrA_HopperKeyOld : USINT;
	ExtrB_HopperKeyOld : USINT;
	LubricCheckA : Lubricate_Check_typ;
	LubricCheckB : Lubricate_Check_typ;
	LubricCheckVisu : Lubricate_Check_typ;
	MotorSpeedA : speedAdjust_typ;
	MotorSpeedB : speedAdjust_typ;
	MotorSpeedVisu : speedAdjust_typ;
	tExtrA_OnNormal : REAL;
	tExtrB_OnNormal : REAL;
	tExtrV_OnNormal : REAL;
	cntExtruderStopDelay : UDINT;
END_VAR
```

### Program Logical/machine/pump (ANSIC, version 1.00.0) - pump,extruder on off

#### pump.c
```c
/********************************************************************
 * COPYRIGHT --  B&R China
 ********************************************************************
 * Program: power
 * File: power.c
 * Author: lijianjun
 * Created: March 06, 2013
 ********************************************************************
 * Implementation of program power --- pump  control
 ********************************************************************/

#include <bur/plctypes.h>

#ifdef _DEFAULT_INCLUDES
#include <AsDefault.h>
#endif

#include "pic_id.h"
/**************************************************************************************
** 					               include user files								          **
**************************************************************************************/
#include "edge.h"               /*edge function                         */
#include "keyap2100.h"
//#include "keyap880.h"
#include "pic_id.h"

/**************************************************************************************
     	        	           I N I T U P  O F   T H E   T A S K
**************************************************************************************/
_INIT void init ( void )
{
	RTInfo_Task.enable = 1;
	RTInfo(&RTInfo_Task);

	tTask = RTInfo_Task.cycle_time/1000.0/1000.0;		/*  from us ---> s  */

	AccuStopCounter = 0;
	AccuStopDelay   = 0;

	OilPumpOnDelay  = 0;
	OilPumpOffDelay = 0;

	HighSafeV_Keep  = 0;
	LowerSafeV_Keep = 0;

	//   gMachineOut.HeatPower = 1;

	tParisonOnDelay = 0;
} /* end of _INIT */

/**************************************************************************************
        				   C Y C L I C   P A R T   O F   T H E   T A S K
**************************************************************************************/

_CYCLIC void cyclic ( void )
{
	tParisonOnDelay = tParisonOnDelay + tTask;
	if(tParisonOnDelay > 10000)tParisonOnDelay = 1000;

	gMachineInfo.Mark = gThickIO.Out.MarkPulse;

	gMachineFix.Pump.PumpOnDealy  = 10;			/*  default value 0.1s */
	gMachineFix.Pump.AccuOffDealy = 10;			/*  default value 0.1s */
	gMachineFix.Pump.PumpOffDealy = 10;			/*  default value 0.1s */

	/* ----------------------- 油泵启动，加热电源 ------------------------- */
	if(1 == gMachineIn.MainControl && gPanelObj.GetPicture != PIC_INIT && (gPanelObj.GetPicture != PIC_SCREEN_SAVE))
	{
		if(1 == EDGEPOS(gPanelObj.KeyMatric[S$KEYMATRIX_PENU_VALVE],PKeyMatric[S$KEYMATRIX_PENU_VALVE]))
		{
			gMachineOut.PneumaticValve = !gMachineOut.PneumaticValve;
		}

		if(1 == EDGEPOS(gPanelObj.KeyMatric[S$KEYMATRIX_HEAT_POWER],PKeyMatric[S$KEYMATRIX_HEAT_POWER]))
		{
			gMachineOut.HeatPower = !gMachineOut.HeatPower;
			gT_Par.GrpSwh.OnOff[0] =  gMachineOut.HeatPower; //1226 ipis
			gT_Par.GrpSwh.PreOnOff[0]=0;
		}

		/*  --------------------- Cooling pump --------------------- */
		if(1 == EDGEPOS(gPanelObj.KeyMatric[S$KEYMATRIX_COOLING_PUMP],PKeyMatric[S$KEYMATRIX_COOLING_PUMP]))
			{
			if(1 == gMachineOut.OilCoolingPump)
			{
				gMachineOut.OilCoolingPump = 0;
			}
			else
			{
				if(1 == gMachineIn.CoolingPumpEnable)
				{
					gMachineOut.OilCoolingPump = 1;
				}
				else
				{
					gImply.CoolingPumpCondition = 1;
				}
			}
		}

		if ( 1 == gMachineFix.ExtruderA.LinkWithMode)
		{
			/*  --------------------- Parison pump && Extuder A --------------------- */
			if( 1 == EDGEPOS(gPanelObj.KeyMatric[S$KEYMATRIX_PARISON_PUMP],PKeyMatric[S$KEYMATRIX_PARISON_PUMP])
				||1 == EDGEPOS(gPanelObj.KeyMatric[S$KEYMATRIX_EXTRUDER_A_ABB],PKeyMatric[S$KEYMATRIX_EXTRUDER_A_ABB]))
				{
				if (0==gExtruderTempLow_HMIFlag)  //ipis0213
				{
					if (0==gMachineInfo.bLoweringFlag)
					{
						if(tParisonOnDelay > gT_Par.Fix.tCheck)
						{
							if(1 == gMachineOut.ParisonPump)
							{
								gMachineOut.ParisonPump = 0;
							}
							else
							{
								if(1 == gExtruderA.Status.OnProtected )  //from  extruder A switch on delay
								{
									if(1 == gMachineIn.ParisonPumpEnable)
									{
										gMachineOut.ParisonPump = 1;
										gThickIO.InitPower = 1;
									}
									else
									{
										gImply.ParisonPumpCondition = 1;
									}
								}
								else
								{
									gImply.ExtrA_OnDelay = 1;
								}
							}
						}
					}
					else
					{
						gImply.TempLoweringEnable =1;
					}
				}
				else
				{
					gImply.TempLow =1;
				}
			}
		}
		else
		{
			/*  --------------------- Parison pump --------------------- */
			if( 1 == EDGEPOS(gPanelObj.KeyMatric[S$KEYMATRIX_PARISON_PUMP],PKeyMatric[S$KEYMATRIX_PARISON_PUMP]))
				{
				if(tParisonOnDelay > gT_Par.Fix.tCheck)
				{
					if(1 == gMachineOut.ParisonPump)
					{
						gMachineOut.ParisonPump = 0;
					}
					else
					{
						if(1 == gMachineIn.ParisonPumpEnable)
						{
							gMachineOut.ParisonPump = 1;
							gThickIO.InitPower = 1;
						}
						else
						{
							gImply.ParisonPumpCondition = 1;
						}
					}
				}
			}
		}

		/*  --------------------- Main pump --------------------- */
		if(1 == EDGEPOS(gMachineIn.OilPumpOnoff,PMachineIn.OilPumpOnoff))
		{
			if((0 == OilPumpOnCounter) && (0 == OilPumpOffCounter))
			{
				if(1 == gMachineOut.OilPump)
				{
					gMachineOut.OilPump = 0;

					AccuStopCounter   = gMachineFix.Pump.AccuOffDealy/2;			/*  off delay     */
					OilPumpOffCounter = gMachineFix.Pump.PumpOffDealy/2;
				}
				else
				{
					OilPumpOnCounter = gMachineFix.Pump.PumpOnDealy/2;
					gMachineOut.OilPumpContactor = 1;                           /*  pump contactor */
				}
			}
		}/* if(1 == EDGEPOS(gMachineIn.OilPumpOnoff,PMachineIn.OilPumpOnoff)) */
	}/* if(1 == gMachineIn.MainControl && gPanelObj.GetPicture != PIC_INIT && gPanelObj.GetPicture != PIC_SCREEN_SAVE) */

	/*  油泵延时启动  */
	if(OilPumpOnCounter > 0)OilPumpOnCounter--;
	OilPumpOnDelay = (OilPumpOnCounter * 2)/10;
	if(OilPumpOnCounter == 1 && 1 == gMachineOut.OilPumpContactor)
	{
		if(1 == gMachineIn.OilPumpEnable && 1 == gMachineIn.CoolingPumpRunning)
		{
			gMachineOut.OilPump = 1;
			gMachineOut.AccuRelieveValve = 1;
		}
		else
		{
			if(0 == gMachineIn.OilPumpEnable)gImply.MainPumpCondition = 1;
			if(0 == gMachineIn.CoolingPumpRunning)gImply.CoolingPumpNotOn = 1;
		}
	}

	/*  油泵接触器延时关闭  */
	if(OilPumpOffCounter > 0)OilPumpOffCounter--;
	OilPumpOffDelay = (OilPumpOffCounter * 2)/10;
	if(OilPumpOffCounter == 1 && 0 == gMachineOut.OilPump)
	{
		gMachineOut.OilPumpContactor = 0;
	}

	/*  储能卸荷延时  */
	if(AccuStopCounter > 0)AccuStopCounter--;
	AccuStopDelay = (AccuStopCounter * 2)/10;
	if(AccuStopCounter == 1 && 0 == gMachineOut.OilPump)
	{
		gMachineOut.AccuRelieveValve = 0;
	}

	/* ----------------------------- oil pump off ------------------------------- */
	if(0 == gMachineInfo.Calib)
	{
		if(1 == gMachineIn.InstancyStop || 0 == gMachineIn.SafeGate || 1 == gMachineInfo.SafeInStop)
		{
			gMachineOut.OilPump = 0;
			gAlarm.SaftyDoor = !gMachineIn.SafeGate;
		}

		gMachineOut.SafetyGateBypass = 0;
	}
	else
	{
		if(1 == gMachineIn.InstancyStop || 1 == gMachineInfo.SafeInStop)
		{
			gMachineOut.OilPump = 0;
			gMachineOut.SafetyGateBypass = 0;
		}
		else
		{
			/* 允許安全門開時開油泵  */
			if(gPanelObj.GetPicture != PIC_CALIB_CLAMP_LVDT && gPanelObj.GetPicture != PIC_CALIB_CARRIAGE_LVDT && gPanelObj.GetPicture != PIC_CALIB_BLOWPIN_LVDT && gPanelObj.GetPicture != PIC_CALIB_OTHER_LVDT )
			{
				gMachineOut.SafetyGateBypass = 0;
			}
			else
			{
				if(1 == gMachineOut.SafetyGateBypass)
				{

				}
				else if(0 == gMachineIn.SafeGate )
				{

					gAlarm.SaftyDoor = !gMachineIn.SafeGate;
					gMachineOut.OilPump = 0;
				}
			}
		}
	}

	/*  main pump feedback check  */
	//	gMachineIn.OilPumpRunning = gMachineOut.OilPump;/*Sinece we don't have feedback, ingore check signal*/
	//	if(gMachineOut.OilPump != gMachineIn.OilPumpRunning)
	//	{
	//		tMainPumpNormal = tMainPumpNormal + tTask;
	//		if(tMainPumpNormal >= 200.0)tMainPumpNormal = 20.0;
	//
	//		if(tMainPumpNormal >= 10.0)
	//		{
	//			gAlarm.OilPumpErr = 1;
	//		}
	//	}
	//	else
	//	{
	//		gAlarm.OilPumpErr = 0;
	//		tMainPumpNormal = 0;
	//	}

	if(1 == gAlarm.OilPumpErr || 0 == gMachineIn.OilPositionNormal || 0 == gMachineIn.OilPumpEnable ||
		0 == gMachineIn.CoolingPumpRunning                          || 0 == gMachineIn.SafeGate)
	{
		if(1 == gMachineOut.OilPump)
		{
			if(0 == gMachineIn.OilPumpEnable)gImply.MainPumpCondition = 1;
			if(0 == gMachineIn.CoolingPumpRunning)gImply.CoolingPumpNotOn = 1;
			if(0 == gMachineIn.SafeGate)gAlarm.SaftyDoor = 1;
			gPROCESS_info.oilpumpStop = 1;   //request manual mode
			gMachineOut.OilPump = 0;
		}
	}

	/*  -------------------- Parison pump off -------------------- */
	/*  Pariosn pump feedback check  */
	gMachineIn.ParisonPumpRunning = gMachineOut.ParisonPump;
	if(gMachineOut.ParisonPump != gMachineIn.ParisonPumpRunning)
	{
		tParisonPumpNormal = tParisonPumpNormal + tTask;
		if(tParisonPumpNormal >= 200.0)tParisonPumpNormal = 20.0;

		if(tParisonPumpNormal >= 10.0)
		{
			gAlarm.ParisonPumpErr = 1;
		}
	}
	else
	{
		gAlarm.ParisonPumpErr = 0;
		tParisonPumpNormal = 0.0;
	}

	if (1 == gMachineInfo.ExtrTLow || 0 == gMachineIn.ParisonPumpEnable || 1 == gAlarm.ParisonPumpErr || 1== gAlarm.ParisonMotorOverload || 0 == gMachineOut.HeatPower
		/*||  (0 == gMachineInfo.IsHeat)*/ || 0 == gT_Par.GrpSwh.OnOff[0]
		|| (gMachineFix.Parison.eActuatorType == ACTUATOR_ELECTRIC &&  ( 1 == gAlarm.ParisonAxisErr || 1 == gAlarm.ParisonNetworkErr)))
	{
		if(1 == gMachineOut.ParisonPump)
		{
			if(1 == gMachineInfo.ExtrTLow)gAlarm.ScrewTempLow = gMachineInfo.ExtrTLow;
			if(0 == gMachineIn.ParisonPumpEnable)gImply.ParisonPumpCondition = 1;
			if(0 == gT_Par.GrpSwh.OnOff[0])gImply.HeatNotOn = 1;
			if(0 == gMachineOut.HeatPower) gImply.HeaterPowerNotOn = 1;
			gMachineOut.ParisonPump = 0;
			gMachineInfo.ParisonPump_ErrStop_LinkWith = 1;  //Extruder Link With Selection
		}
	}

	/* ------------------------ Pump Link With Selection  ---------------------------- */
	/* ----- ParisonPump ----- */
	if(1 == gMachineFix.ExtruderA.LinkWithMode)
	{
		//		if( EDGENEG(gMachineOut.ParisonPump,oldParisonPump_On))
		//		{
		//			gMachineOut.ExtrA_On = 0;
		//		}
		//		else
		if(1 == gMachineInfo.ParisonPump_ErrStop_LinkWith)
		{
			gMachineInfo.ParisonPump_ErrStop_LinkWith = 0;
			gMachineOut.ExtrA_On = 0;
		}
	}

	oldParisonPump_On = gMachineOut.ParisonPump;
	/*  -------------------- Cooling pump off -------------------- */
	/*  Cooling pump feedback check  */
	//	gMachineIn.CoolingPumpRunning = gMachineOut.OilCoolingPump;
	//	if(gMachineOut.OilCoolingPump != gMachineIn.CoolingPumpRunning)
	//	{
	//		tCoolingPumpNormal = tCoolingPumpNormal + tTask;
	//		if(tCoolingPumpNormal >= 200.0)tCoolingPumpNormal = 20.0;
	//
	//		if(tCoolingPumpNormal >= 10.0)
	//		{
	//			gAlarm.CoolingPumpErr = 1;
	//		}
	//	}
	//	else
	//	{
	//		gAlarm.CoolingPumpErr = 0;
	//		tCoolingPumpNormal = 0.0;
	//	}

	if (0 == gMachineIn.CoolingPumpEnable || 1 == gAlarm.CoolingPumpErr)
	{
		if(1 == gMachineOut.OilCoolingPump)
		{
			gMachineOut.OilCoolingPump = 0;
			if (0 == gMachineIn.CoolingPumpEnable)gImply.CoolingPumpCondition = 1;
		}
	}

	/* Oil cooling pump auto cooling  -> OilCoolingValve */
	if(!gMachineFix.OilCooling.OilTempCoolingStart)gMachineFix.OilCooling.OilTempCoolingStart = 40;
	if(!gMachineFix.OilCooling.OilTempCoolingStop)gMachineFix.OilCooling.OilTempCoolingStop = 35;

	if(gMachineInfo.OilTemp > gMachineFix.OilCooling.OilTempCoolingStart)
	{
		gMachineOut.WaterCooling = 1;
	}

	if(gMachineInfo.OilTemp < gMachineFix.OilCooling.OilTempCoolingStop)
	{
		gMachineOut.WaterCooling = 0;
	}
	gMachineOut.OilCoolingValve = !gMachineOut.WaterCooling;

	/* ------------------------ hot cutter heating  熱切刀 DO -------------------------- */
	//	if(1 == EDGEPOS(gMachineIn.Key.HotCutter,PMachineIn.Key.HotCutter))
	//	{
	//		gMachineOut.CutterHeating = !gMachineOut.CutterHeating;
	//	}
	//
	//	if(1 == gMachineOut.CutterHeating)
	//	{
	//		if(gMachineOut.CutterHeating != gMachineIn.HotCutterNormal)
	//		{
	//			tCutterHeatNormal = tCutterHeatNormal + tTask;
	//			if(tCutterHeatNormal >= 200.0)tCutterHeatNormal = 20.0;
	//		}
	//		else
	//		{
	//			tCutterHeatNormal = 0;
	//		}
	//	}
	//	else
	//	{
	//		tCutterHeatNormal = 0;
	//	}
	//
	//	if(tCutterHeatNormal >= 10.0)
	//	{
	//		gAlarm.CutterHeatNormal = 1;  /*  熱切刀加熱異常  */
	//		if(gMachineOut.CutterHeating != 0)gMachineOut.CutterHeating = 0;
	//	}
	//	else
	//	{
	//		gAlarm.CutterHeatNormal = 0;
	//	}

	gMachineOut.LowerRelieveValve  = gMachineOut.OilPump;
	gMachineOut.HigherRelieveValve = gMachineOut.OilPump;

	if(1 == gMachineIn.LowerPressureHigh && 0 == gMachineIn.LowerPressureLow)
	{
		gMachineOut.LowerRelieveValve = 0;
	}

	/* ----------------- high pressure/low pressure enable valve --------------- */
	if(0 == gMachineInfo.Calib)
	{
		gMachineOut.HighPressureEnable = !gMachineIn.InstancyStop | gMachineIn.SafeGate | gMachineIn.OilPumpRunning | !gMachineInfo.SafeInStop;
		gMachineOut.LowPressureEnable  = !gMachineIn.InstancyStop | gMachineIn.SafeGate | gMachineIn.OilPumpRunning | !gMachineInfo.SafeInStop;
	}
	else
	{
		gMachineOut.HighPressureEnable = !gMachineIn.InstancyStop | gMachineIn.OilPumpRunning | !gMachineInfo.SafeInStop;
		gMachineOut.LowPressureEnable  = !gMachineIn.InstancyStop | gMachineIn.OilPumpRunning | !gMachineInfo.SafeInStop;
	}

	/*  -------------------------Safe Calib Pressure --------------------- */
	if(1 == gMachineIn.LMold.SafeGate && 1 == gMachineIn.RMold.SafeGate)
	{
		if(gMachineOut.OilPump == 1)
		{
			if(0 == gMachineInfo.Calib)
			{
				gMachineOut.SafeCalibPressure      = 1;
			}
			else
			{
				gMachineOut.SafeCalibPressure      = gMachineIn.CalibMode;
			}
		}
		else
		{
			gMachineOut.SafeCalibPressure     = 0;
		}
	}
	else
	{
		gMachineOut.SafeCalibPressure      = gMachineOut.OilPump;
	}

	gMachineOut.InerloclResetEnable =  gMachineIn.HydPressureSW | gMachineIn.PnePressureSW;

	/* ----------------------------- Safety reset lamp  ------------------------------- */
	cntFlasher++;
	if(cntFlasher >= 20000)cntFlasher=0;

	if(0 == gMachineIn.InstancyStop && 1 == gMachineIn.SafeGate && 0 == gMachineInfo.SafeInStop)
	{
		gMachineOut.InerloclResetLed = 1;
	}
	else
	{
		if(1 == gMachineIn.InstancyStop || 0 == gMachineIn.SafeGate  || 1 == gMachineInfo.SafeInStop)
		{
			/* lamp falsher   */
			if((cntFlasher%100) < 50)
			{
				gMachineOut.InerloclResetLed = 1;
			}
			else
			{
				gMachineOut.InerloclResetLed = 0;
			}
		}
		else
		{
			gMachineOut.InerloclResetLed = 0;
		}
	}/* if(0 == gMachineIn.InstancyStop && 1 == gMachineIn.SafeGate) */

	gThickIO.BtnPowerOn = gMachineOut.ParisonPump;

	if(1 == EDGEPOS(gPanelObj.KeyMatric[S$KEYMATRIX_MAIN_PUMP],PKeyMatric[S$KEYMATRIX_MAIN_PUMP]))
		{
		if(1 == gMachineIn.MainControl && gPanelObj.GetPicture != PIC_INIT && gPanelObj.GetPicture != PIC_SCREEN_SAVE)
		{
			if (1 == gMachineIn.AccuChargeON && 0 == gMachineOut.OilPump)
			{/*2020.08.27 Chaoi*/
				gAlarm.AccuChargeRPressure = 1;
			}
			else
			{
				if(  1 == gMachineInfo.DriverNetworkPhaseReady  )
				{
					if( 1 == gMachineIn.SafeGate )
					{
						if(0 == gMachineOut.OilPump)
						{
							gMachineOut.OilPump = 1;

							RMold.ExtrLift.InitPower = 1;

							LMold.Clamp.InitPower = 1;
							RMold.Clamp.InitPower = 1;

							LMold.Carriage.InitPower = 1;
							RMold.Carriage.InitPower = 1;

							LMold.BlowPin.InitPower = 1;
							RMold.BlowPin.InitPower = 1;

							LMold.BlowPin2.InitPower = 1;
							RMold.BlowPin2.InitPower = 1;

							LMold.Robot.Transfer.InitPower = 1;
							RMold.Robot.Transfer.InitPower = 1;

							LMold.Robot.UpDn.InitPower = 1;
							RMold.Robot.UpDn.InitPower = 1;

							LMold.Sensor.UpDn.InitPower = 1;
							RMold.Sensor.UpDn.InitPower = 1;
						}
						else
						{
							if((0.0 == LMold.Clamp.v_set   ) && (0.0 == RMold.Clamp.v_set   ) &&
								(0.0 == LMold.Carriage.v_set) && (0.0 == RMold.Carriage.v_set) &&
								(0.0 == LMold.BlowPin.v_set ) && (0.0 == RMold.BlowPin.v_set )&&
								(0.0 == LMold.BlowPin2.v_set ) && (0.0 == RMold.BlowPin2.v_set ))
							{
								gMachineOut.OilPump = 0;
							}
						}
					}
					else
					{
						gImply.SafeGate = !gMachineIn.SafeGate;
					}

				}
				else
				{
					gImply.DriverNetworkPhaseNotReady = !gMachineInfo.DriverNetworkPhaseReady;
				}
			}
		}
	}

	RMold.ExtrLift.BtnPowerOn = gMachineOut.OilPump;

	LMold.Clamp.BtnPowerOn = gMachineOut.OilPump;
	RMold.Clamp.BtnPowerOn = gMachineOut.OilPump;

	LMold.Carriage.BtnPowerOn = gMachineOut.OilPump;
	RMold.Carriage.BtnPowerOn = gMachineOut.OilPump;

	LMold.BlowPin.BtnPowerOn = gMachineOut.OilPump;
	RMold.BlowPin.BtnPowerOn = gMachineOut.OilPump;

	LMold.BlowPin2.BtnPowerOn = gMachineOut.OilPump;
	RMold.BlowPin2.BtnPowerOn = gMachineOut.OilPump;

	LMold.Robot.UpDn.BtnPowerOn =  gMachineOut.OilPump;
	RMold.Robot.UpDn.BtnPowerOn =  gMachineOut.OilPump;

	LMold.Robot.Transfer.BtnPowerOn =  gMachineOut.OilPump;
	RMold.Robot.Transfer.BtnPowerOn =  gMachineOut.OilPump;

	LMold.Sensor.UpDn.BtnPowerOn = gMachineOut.OilPump;
	RMold.Sensor.UpDn.BtnPowerOn = gMachineOut.OilPump;

	gMachineOut.CarriagePower = gMachineOut.OilPump;
	gMachineOut.ClampPower    = gMachineOut.OilPump;
	gMachineOut.BlowPinPower  = gMachineOut.OilPump;

	/* ----------------------------- safety gate lock ------------------------------- */
	if(0 == gMachineOut.OilPump && 1 == gMachineIn.PnePressureSW)
	{
		gMachineOut.SafetyGateUnlock = 1;
	}
	else
	{
		gMachineOut.SafetyGateUnlock = gMachineInfo.Calib;
	}

	/* ----------------------------- waste belt control ------------------------------- */
	if(0 == gMachineInfo.Calib)
	{
		if(0 == StepWasteBelt)StepWasteBelt = 10;
	}
	else
	{
		StepWasteBelt = 0;
	}

	switch(StepWasteBelt)
	{
		case 0:
			gMachineOut.WasteBelt  = 0;
			gMacTimer.WasteBelt.IN = 0;
			break;

		case 10:
			if(gMachinePara.WateBeltOffTime > 0.0)
			{
				gMacTimer.WasteBelt.IN = 1;
				gMacTimer.WasteBelt.PT = (UDINT)(gMachinePara.WateBeltOffTime * 100);
				StepWasteBelt = 20;
			}
			else
			{
				StepWasteBelt = 30;
			}
			break;

		case 20:
			gMachineOut.WasteBelt = 0;

			if(1 == gMacTimer.WasteBelt.Q)
			{
				gMacTimer.WasteBelt.IN = 0;
				StepWasteBelt = 30;
			}
			break;

		case 30:
			gMacTimer.WasteBelt.IN = 0;
			StepWasteBelt = 40;
			break;

		case 40:
			if(gMachinePara.WateBeltOnTime > 0.0)
			{
				gMacTimer.WasteBelt.IN = 1;
				gMacTimer.WasteBelt.PT = (UDINT)(gMachinePara.WateBeltOnTime * 100);
				StepWasteBelt = 50;
			}
			else
			{
				StepWasteBelt = 60;
			}
			break;

		case 50:
			gMachineOut.WasteBelt = 1;

			if(1 == gMacTimer.WasteBelt.Q)
			{
				gMacTimer.WasteBelt.IN = 0;
				StepWasteBelt = 60;
			}
			break;

		case 60:
			gMachineOut.WasteBelt  = 0;
			gMacTimer.WasteBelt.IN = 0;
			StepWasteBelt = 10;
			break;
	}/* switch(StepWasteBelt) */

	/* ----------------------------- key edge ------------------------------- */
	PKeyMatric[S$KEYMATRIX_HEAT_POWER]  = gPanelObj.KeyMatric[S$KEYMATRIX_HEAT_POWER];
		PKeyMatric[S$KEYMATRIX_PENU_VALVE]  = gPanelObj.KeyMatric[S$KEYMATRIX_PENU_VALVE];

		PMachineIn = gMachineIn;
	NMachineIn = gMachineIn;

} /* end of _CYCLIC */
```

#### pump.var
```iecst
VAR
	tTask : REAL := 0.0;
	tParisonOnDelay : REAL;
	StepWasteBelt : UINT;
	tCutterHeatNormal : REAL;
	tMainPumpNormal : REAL;
	tParisonPumpNormal : REAL;
	tCoolingPumpNormal : REAL;
	RTInfo_Task : RTInfo := (0);
	PMachineIn : Machine_In_typ;
	NMachineIn : Machine_In_typ;
	PKeyMatric : ARRAY[0..MAX_KEY_COUNT] OF USINT;
	cntFlasher : UDINT;
	AccuStopCounter : UDINT;
	AccuStopDelay : UDINT;
	OilPumpOnDelay : UINT;
	OilPumpOffDelay : UINT;
	OilPumpOnCounter : UINT;
	OilPumpOffCounter : UINT;
	HighSafeV_Keep : UDINT;
	LowerSafeV_Keep : UDINT;
	oldParisonPump_On : USINT;
END_VAR
```

- pic_id.h (reference to Logical/GlobalIncludes/pic_id.h)

### Program Logical/machine/mac_lubr (ANSIC, version 1.00.0) - machine lubrication

- edge.h (reference to Logical/GlobalIncludes/edge.h)

#### lubricate.c
```c
/********************************************************************
 * COPYRIGHT --  B&R China
 ********************************************************************
 * Program: lubricate
 * File: lubricate.c
 * Author: lijianjun
 * Created: March 06, 2013
 ********************************************************************
 * Implementation of program lubricate --- oil lubrication control
 ********************************************************************/

#include <bur/plctypes.h>

#ifdef _DEFAULT_INCLUDES
	#include <AsDefault.h>
#endif

#include "edge.h"               /*  edge function  */
#include "keyap2100.h"
//#include "keyap880.h"

/**************************************************************************************
     	        		I N I T U P  O F   T H E   T A S K
**************************************************************************************/
void _INIT lubr_init(void)
{
	TimeStep  = 0;
   LubricateStep  = 0;
   LMold.Lubricate.Step = 0;
   RMold.Lubricate.Step = 0;
	Count = 0;
}  /* end of _INIT */
/**************************************************************************************
****				C Y C L I C   P A R T   O F   T H E   T A S K  				   ****
**************************************************************************************/
void _CYCLIC lubr_cyclic(void)
{
	/* -------------- Machine running time -------------- */
	Count++;
	if(Count >=300000)Count=0;
	if(0 == Count%3000)
	{
		gMachineWorkTime++;
	}

   /* -------------- Machine yield -------------- */
   if(gMachinePara.DieheadNum < 1)gMachinePara.DieheadNum = 1;
   gMachineInfo.Yield = gMachineInfo.CycleTimes * gMachinePara.DieheadNum;

	if(1 == gMachineInfo.Auto)
	{
		if(1 == LMold.Option.Enable && 1 == RMold.Option.Enable)
		{
			if(LMold.TimeDis.CycleAlarmTime != 0 && RMold.TimeDis.CycleAlarmTime != 0)
			{
				gMachineInfo.Yield_H = 3600.0 * 100 * 4/(LMold.TimeDis.CycleAlarmTime + RMold.TimeDis.CycleAlarmTime) * gMachinePara.DieheadNum;
			}
			else
			{
				gMachineInfo.Yield_H = 0;
			}
		}
		else if(1 == LMold.Option.Enable && 0 == RMold.Option.Enable)
		{
			if(LMold.TimeDis.CycleAlarmTime != 0)
			{
				gMachineInfo.Yield_H = 3600.0 * 100/LMold.TimeDis.CycleAlarmTime * gMachinePara.DieheadNum;
			}
			else
			{
				gMachineInfo.Yield_H = 0;
			}
		}
		else if(0 == LMold.Option.Enable && 1 == RMold.Option.Enable)
		{
			if(RMold.TimeDis.CycleAlarmTime != 0)
			{
				gMachineInfo.Yield_H = 3600.0 * 100 /RMold.TimeDis.CycleAlarmTime * gMachinePara.DieheadNum;
			}
			else
			{
				gMachineInfo.Yield_H = 0;
			}
		}
	}

   if((gMachinePara.StopYield > 0) && (1 == gMachinePara.bReachYieldStop))
   {
      if((gMachineInfo.Yield >= gMachinePara.StopYield) && (1 == gMachineInfo.Auto) /*&& (0==gMachineInfo.CycleTimeCounReach)*/)
      {
      //   gPROCESS_info.semi_auto = 1;
			gAlarm.CycleTimeCounReach =1;
			gMachineInfo.CycleTimeCounReach = 1;
			gPanelObj.RKeyMatric[S$KEYMATRIX_AUTO_STOP] = 1;
			gDisableAll_HMI = 1;
			//			gMachineIn.AutoStop =1;   //ipis0131
      }
   }
//	if (0==gAlarm.CycleTimeCounReach)
//	{
//		CycleTimeReachFlag =0;
//	}

//	if((gMachinePara.StopYield > 0) && (0 == gMachinePara.bReachYieldStop) &&(0==gAlarm.CycleTimeCounReach)) //ipis0129
//	{
//		if((gMachineInfo.Yield >= gMachinePara.StopYield) && (1 == gMachineInfo.Auto) &&( gCycleTimesOld==gCycleTimes ))
//		{
//
//			CycleTimeReachFlag =1;
//
//		}
//	}
//	else
//	{
//		CycleTimeReachFlag =0;
//	}
//
//	if (EDGEPOS(CycleTimeReachFlag,PCycleTimeReachFlag))
//	{
//		gAlarm.CycleTimeCounReach =1;
//	}

	if (1==bCycleTimeReset)
	{
		gCycleTimes=0;
		gCycleTimesL =0;
		gCycleTimesR =0;
	}
	gMachineInfo.CycleTimes  = gCycleTimes;
	gMachineInfo.CycleTimesL = gCycleTimesL;
	gMachineInfo.CycleTimesR = gCycleTimesR;

	if (1 == bBatchDoneCountReset)
	{
		bBatchDoneCountReset = 0;
		gBatchInfo.Batch = 0;
		gBatchInfo.BatchDoneCount = 0;
	}

   /* -------------- Default lubrication time -------------- */
	if(gMachineFix.Lubrication.LubrPumpWorkTime == 0)gMachineFix.Lubrication.LubrPumpWorkTime = 5;
	if(gMachineFix.Lubrication.LubrPumpStopTime == 0)gMachineFix.Lubrication.LubrPumpStopTime = 6000;
   if(gMachineFix.Lubrication.SetCycleTimes == 0   )gMachineFix.Lubrication.SetCycleTimes = 2000;

   /* ---------------- Start lubrication ---------------- */
	if(1 == EDGEPOS(gMachineOut.OilPump,OilPump))
	{
      if(1 == gUserFix_new.bTimeLubricate)
      {
         if(gMachineFix.Lubrication.LubrPumpWorkTime != 0 && gMachineFix.Lubrication.LubrPumpStopTime != 0)
         {
            TimeStep = 100;  /* first stop time then work time */
         }
         else
         {
            gAlarm.LubrTimeZero = 1;
         }
      }
	}

	if(0 == gMachineOut.OilPump)
	{
		TimeStep = 0;
	}

	if(1 == gMachineIn.LubriFilter || 1 == gMachineIn.LubriOverload)
	{
		TimeStep = 0;
      LubricateStep = 0;
	}

   if(1 == gUserFix_new.bTimeLubricate)     /*  时间控制  */
   {

      /* ---------- step machine control ---------- */
      switch(TimeStep)
      {
         case 0:
            gMacTimer.LubrWork.IN = 0;
            gMacTimer.LubrStop.IN = 0;
			LubrPumpWorkDis = 0;
			LubrPumpStopDis = 0;

            gMachineOut.Lubricate = gPanelObj.KeyMatric[S$KEYMATRIX_LUBRICATION];
            break;

         case 100:
            gMacTimer.LubrWork.IN = 0;
            gMacTimer.LubrStop.IN = 0;
            TimeStep = 200;
            break;

         case 200:
            if(gMachineFix.Lubrication.LubrPumpStopTime != 0)
            {
               gMacTimer.LubrStop.IN = 1;
               gMacTimer.LubrStop.PT = gMachineFix.Lubrication.LubrPumpStopTime * 100 ;
               TimeStep = 300;
            }
            else
            {
               TimeStep = 400;
            }
            break;

         case 300:
            gMachineOut.Lubricate = 0;
            LubrPumpStopDis = gMacTimer.LubrStop.ET/100;

            if(1 == gMacTimer.LubrStop.Q)
            {
               gMachineOut.Lubricate = 0;
               gMacTimer.LubrStop.IN = 0;
               TimeStep = 400;
            }
            break;

         case 400:
            if(gMachineFix.Lubrication.LubrPumpWorkTime != 0)
            {
               gMacTimer.LubrWork.IN = 1;
               gMacTimer.LubrWork.PT = gMachineFix.Lubrication.LubrPumpWorkTime * 100 ;
               TimeStep = 500;
            }
            else
            {
               TimeStep = 600;
            }
            break;

         case 500:
            gMachineOut.Lubricate = 1;
            LubrPumpWorkDis = gMacTimer.LubrWork.ET/100;

            if(1 == gMacTimer.LubrWork.Q)
            {
               gMachineOut.Lubricate = 0;
               gMacTimer.LubrWork.IN = 0;
               TimeStep = 600;
            }
            break;

         case 600:
            TimeStep = 100;
            break;
      }/* switch(Step) */
   }/* if(1 == gUserFix_new.bTimeLubricate) */
   else
   {
      TimeStep = 0;
   }

   /* Lubrication auto start*/
   if((0 ==(gMachineInfo.CycleTimes % gMachineFix.Lubrication.SetCycleTimes))&& (gMachineInfo.CycleTimes != 0))
   {
      if(gMachineInfo.CycleTimes != OldCycleTimes)
      {
         if(0 == gUserFix_new.bTimeLubricate)LubricateStep = 100;
      }
   }

   OldCycleTimes = gMachineInfo.CycleTimes;

   if(0 == gUserFix_new.bTimeLubricate)     /*  次数控制  */
   {
      /* step machine control */
      switch(LubricateStep)
      {
         case 0:
            gMacTimer.LubrWork.IN = 0;
            gMachineOut.Lubricate = gPanelObj.KeyMatric[S$KEYMATRIX_LUBRICATION];
            LubrPumpWorkDis = 0;
            break;

         case 100:
            gMacTimer.LubrWork.IN = 1;
            gMacTimer.LubrWork.PT = gMachineFix.Lubrication.LubrPumpWorkTime * 100;
            LubricateStep  = 200;
            break;

         case 200:
            gMachineOut.Lubricate = 1;
            LubrPumpWorkDis = gMacTimer.LubrWork.ET/100;
            if(1 == gMacTimer.LubrWork.Q)
            {
               gMachineOut.Lubricate = 0;
               LubrPumpWorkDis  = 0;
               gMacTimer.LubrWork.IN = 0;
               LubricateStep  = 300;
            }
            break;

         case 300:
            gMachineOut.Lubricate = 0;
            LubricateStep = 0;
            break;
      }/* switch(LubricateStep) */
   }/* if(0 == gUserFix_new.bTimeLubricate) */
   else
   {
      LubricateStep = 0;
   }

   /*  left mold manual button start  */
   if(1 == gPanelObj.KeyMatric[S$KEYMATRIX_LUBRICATION])
   {
		if((0 == RightOption) && (1 == LeftOption))
		{
			if(0 == LMold.Lubricate.Step)LMold.Lubricate.Step = 100;
		}
   }

   /* left mold auto start*/
   if((0 ==(gMachineInfo.CycleTimesL % gMachineFix.Lubrication.SetCycleTimes))&& (gMachineInfo.CycleTimesL != 0))
   {
      if(gMachineInfo.CycleTimesL != OldCycleTimesL)
      {
         if(1 == LMold.Option.Enable)LMold.Lubricate.Step = 100;
      }
   }

   OldCycleTimesL = gMachineInfo.CycleTimesL;

   /* step machine control */
   switch(LMold.Lubricate.Step)
   {
      case 0:
         LMold.Lubricate.Timer.IN = 0;
         gMachineOut.LMold.Lubricate = 0;
         LubrPumpWorkDisL = 0;
         break;

      case 100:
         LMold.Lubricate.Timer.IN = 1;
         LMold.Lubricate.Timer.PT = gMachineFix.Lubrication.LubrPumpWorkTime * 100;
         LMold.Lubricate.Step  = 200;
         break;

      case 200:
         gMachineOut.LMold.Lubricate = 1;
         LubrPumpWorkDisL = LMold.Lubricate.Timer.ET/100;
         if(1 == LMold.Lubricate.Timer.Q)
         {
            LubrPumpWorkDisL  = 0;
            LMold.Lubricate.Timer.IN = 0;
            LMold.Lubricate.Step  = 300;
         }
         break;

      case 300:
         gMachineOut.LMold.Lubricate = 0;
         if(0 == gPanelObj.KeyMatric[S$KEYMATRIX_LUBRICATION])
         {
            gMachineOut.LMold.Lubricate = 0;
            LMold.Lubricate.Step = 0;
         }
         break;
   }/* switch(LMold.Lubricate.Step) */

   /*  Right mold manual button start  */
   if(1 == gPanelObj.KeyMatric[S$KEYMATRIX_LUBRICATION])
   {
		if((1 == RightOption) && (0 == LeftOption))
		{
			if(0 == RMold.Lubricate.Step)RMold.Lubricate.Step = 100;
		}
   }

   /* right mold */
   if((0 ==(gMachineInfo.CycleTimesR % gMachineFix.Lubrication.SetCycleTimes))&& (gMachineInfo.CycleTimesR != 0))
   {
      if(gMachineInfo.CycleTimesR != OldCycleTimesR)
      {
         if(1 == RMold.Option.Enable)RMold.Lubricate.Step = 100;
      }
   }

   OldCycleTimesR = gMachineInfo.CycleTimesR;

   /* step machine control */
   switch(RMold.Lubricate.Step)
   {
      case 0:
         RMold.Lubricate.Timer.IN = 0;
         gMachineOut.RMold.Lubricate = 0;
         LubrPumpWorkDisR = 0;
         break;

      case 100:
         RMold.Lubricate.Timer.IN = 1;
         RMold.Lubricate.Timer.PT = gMachineFix.Lubrication.LubrPumpWorkTime * 100;
         RMold.Lubricate.Step  = 200;
         break;

      case 200:
         gMachineOut.RMold.Lubricate = 1;
         LubrPumpWorkDisR = RMold.Lubricate.Timer.ET/100;
         if(1 == RMold.Lubricate.Timer.Q)
         {
            LubrPumpWorkDisR  = 0;
            RMold.Lubricate.Timer.IN = 0;
            RMold.Lubricate.Step  = 300;
         }
         break;

      case 300:
         gMachineOut.RMold.Lubricate = 1;
         if(0 == gPanelObj.KeyMatric[S$KEYMATRIX_LUBRICATION])
         {
            gMachineOut.RMold.Lubricate = 0;
            RMold.Lubricate.Step = 0;
         }
         break;
   }/* switch(RMold.Lubricate.Step) */

}  /* end of _CYCLIC */
```

#### mac_lubr.var
```iecst
VAR
	TimeStep : UINT;
	Count : UDINT;
	LubrPumpWorkDisL : UDINT;
	LubrPumpWorkDisR : USINT;
	LubrPumpWorkDis : UDINT;
	LubrPumpStopDis : UDINT;
	OilPump : USINT;
	LubricateStep : UDINT;
	OldCycleTimes : UDINT;
	OldCycleTimesL : UDINT;
	OldCycleTimesR : UDINT;
	CycleTimeReachFlag : USINT;
	PCycleTimeReachFlag : USINT;
	bCycleTimeReset : BOOL;
	bBatchDoneCountReset : USINT;
END_VAR
```

- keyap880.h (reference to Logical/GlobalIncludes/keyap880.h)

### Program Logical/machine/oil_accu (ANSIC, version 1.00.0) - oil accumulator control

#### oil_accu.c
```c
/********************************************************************
 * COPYRIGHT --  B&R China
 ********************************************************************
 * Program: oil_accu
 * File: oil_accu.c
 * Author: lijianjun
 * Created: March 06, 2013
 ********************************************************************
 * Implementation of program oil_accu--- accumulator  control
 ********************************************************************/

#include <bur/plctypes.h>

#ifdef _DEFAULT_INCLUDES
#include <AsDefault.h>
#endif

/**************************************************************************************
     	        		I N I T U P  O F   T H E   T A S K
**************************************************************************************/
_INIT void init ( void )
{
	/* ----- get task cycle time ----- */
	RTInfo_Task.enable = 1;
	RTInfo(&RTInfo_Task);

	tTask = RTInfo_Task.cycle_time/1000.0/1000.0;		/*  from us ---> s  */

	ChargeState = 0;
} /* end of _INIT */

 /*************************************************************************************
        				C Y C L I C   P A R T   O F   T H E   T A S K
**************************************************************************************/
_CYCLIC void cyclic ( void )
{
	/*  ------------ 设定值问题 ------------ */
	if(0.0 == gMachineFix.OilAccu.AccuTimeout)gMachineFix.OilAccu.AccuTimeout = 300.0;             /*   s   */
	if(0.0 == gMachineFix.OilAccu.AccuPressureStart)gMachineFix.OilAccu.AccuPressureStart = 70.0;  /*  bar  */
	if(0.0 == gMachineFix.OilAccu.AccuPressureStop)gMachineFix.OilAccu.AccuPressureStop = 90.0;    /*  bar  */
	if(0.0 == gMachineFix.OilAccu.AccuPressure10V)gMachineFix.OilAccu.AccuPressure10V = 200.0;     /*  bar  */
	if(0.0 == gMachineFix.OilAccu.AccuFlow) gMachineFix.OilAccu.AccuFlow	= 0.0; /*Perstange*/

	if(gMachineFix.OilAccu.AccuPressureStop < gMachineFix.OilAccu.AccuPressureStart)
	{
		gMachineFix.OilAccu.AccuPressureStop = gMachineFix.OilAccu.AccuPressureStart + 20;
	}

	/* ------------ 压力传感器问题 ------------ */
	if(gMachineFix.OilAccu.AccuPressure10V != 0)
	{
		if(gMachineFix.OilAccu.AccuPressure10V == gMachineInfo.OilAccuPressure)
		{
			/*gAlarm.AccuSensorError = 1;*/
		}
		else
		{
			gAlarm.AccuSensorError = 0;
		}
	}
	else
	{
		gAlarm.AccuSensorError = 0;
	}

	/*Chaoi*/
	gUserPara.OilPumpDelayTime = 3;
	if (1==gMacOption.OilPumpStartMode)
	{
		if (1==gMachineIn.OilPumpOk_DI)
		{
			if (OilPumpDelayTime >= gUserPara.OilPumpDelayTime)
			{
				gMachineInfo.OilPumpDelayDone =1;
			}
			else
			{
				OilPumpDelayTime = OilPumpDelayTime+tTask;
			}
		}
		else
		{
			gMachineInfo.OilPumpDelayDone =0;
			OilPumpDelayTime =0;
		}
	}
	else
	{
		gMachineInfo.OilPumpDelayDone = 1;
		OilPumpDelayTime =0;
	}

	/* -------------------------------------------- */
	/* ----------------系統蓄壓器------------------ */
	/* ---------------------------------------------*/

	/* ------------ 蓄能器充压控制 ------------ */

	if((1 == gMachineOut.OilPump) && (1 == gMacOption.ACCPumpCharge)
		&& ( 0==gMacOption.OilPumpStartMode || (1==gMachineIn.OilPumpOk_DI && 1==gMachineInfo.OilPumpDelayDone)/*  开启蓄能器  */))
	{
		gMachineOut.ChargeHold	=	gMachineOut.OilPump;/*When Oil pump on then it need hold pressure by enable Hold Valve*/

		gMachineInfo.OilAccuChargeAuto = 0;
		if(gMachineInfo.OilAccuPressure < gMachineFix.OilAccu.AccuPressureStart)
		{
			ChargeFlag = 1;
		}
		else
		{
			ChargeFlag = 0;
		}

		switch (ChargeState)
		{
			case 0:	//StandStill
				gMachineOut.Q_Charge	=	0;
				gMachineOut.P_Charge	=   0;
				gMachineOut.AccuChargeValve = 0;
				timeCount = 0;
				accChargeValveDelayTimeCount = 0;
				accChargeValveTimeCount = 0;
				if(1 == ChargeFlag)
				{
					ChargeState = 1;
				}
				break;

			case 1: //Charging

				accChargeValveDelayTimeCount++;
				if(accChargeValveDelayTimeCount * tTask > gUserFix_new.AccChargeValveDelayTime || 1 == accChargeValveDelayDoneOnce )
				{
					accChargeValveDelayDoneOnce = 1;

					gMachineOut.AccuChargeValve	= 1;
					gMachineOut.Q_Charge		= gMachineFix.OilAccu.AccuFlow;
					gMachineOut.P_Charge		= gMachineFix.OilAccu.AccuChargePressure;
					timeCount ++;
					accChargeValveTimeCount ++;
					if(timeCount * tTask > gMachineFix.OilAccu.AccuTimeout)
					{
						//				gAlarm.AccuChargeError = 1;
					}
				}

				if(gMachineInfo.OilAccuPressure > gMachineFix.OilAccu.AccuPressureStop)
				{
					ChargeState = 0;
				}

				break;

		}

		RelieveCount = 15000;   /* time = 15000 * tTask this task means 300s */

	}
	else
	{
		ChargeState = 0;
		timeCount = 0;
		accChargeValveDelayTimeCount = 0;
		accChargeValveDelayDoneOnce = 0;
		gMachineOut.AccuChargeValve = 0;
		gMachineOut.Q_Charge	=	0;
		gMachineOut.P_Charge	=	0;
		gMachineOut.ChargeHold = 0;/*Reset valve*/
		if(RelieveCount > 0)RelieveCount--;

		if(1 == RelieveCount)
		{
			if(gMachineInfo.OilAccuPressure > 20)
			{
				/*gAlarm.AccuRelieveError = 1;*/
			}
		}
	}/* if(1 == gMachineOut.OilPump)*/

	oldChargeState = ChargeState;
	chargeTime = timeCount * tTask;
	accChargeValveDelayTime = accChargeValveDelayTimeCount * tTask;
	accChargeValveTime = accChargeValveTimeCount * tTask;

	//	gMachineOut.AccuChargeValve = gMachineIn.OilPumpRunning;

	/* ------------ 蓄能器压力可以 ------------ */
	if(gMachineInfo.OilAccuPressure > gMachineFix.OilAccu.AccuPressureStart)
	{
		gMachineInfo.IsAccuOK = 1;
	}
	else
	{
		gMachineInfo.IsAccuOK = 0;
	}

	/* -------------------------------------------- */
	/* ----------------抬頭蓄壓器------------------ */
	/* -------------------------------------------- */

	/* ------------ 抬頭蓄壓器充压控制 ------------ */

	if((1 == gMachineOut.OilPump) && (1 == gMacOption.ACCPumpCharge_Extrlift)
		&& ( 0==gMacOption.OilPumpStartMode || (1==gMachineIn.OilPumpOk_DI && 1==gMachineInfo.OilPumpDelayDone)/*  开启蓄能器  */))
	{
		gMachineOut.ChargeHold_Extrlift	=	gMachineOut.OilPump;/*When Oil pump on then it need hold pressure by enable Hold Valve*/

		if (1 == gMachineInfo.Auto)
		{
			if(1 ==  gMachineInfo.OilAccuChargeAuto_Extrlift && (PRESSURE_OUTPUT_ACC_EXTRLIFT == gMachineFix.ExtrLift.ePressueOutputType && RMold.ExtrLift.Step  == 13000 ) ) /*關模保持結束 && 抬頭結束*/
			{
				gMachineInfo.OilAccuChargeAuto_Extrlift = 0;
				if(gMachineInfo.OilAccuPressure_Extrlift < gMachineFix.OilAccu_Extrlift.AccuPressureStop)
				{
					ChargeFlag_Extrlift = 1;
				}
				else
				{
					ChargeFlag_Extrlift = 0;
				}
			}
		}
		else
		{
			if(( 0 == gMachineFix.Option.bOilAccu_Extrlift_DisChar_Calib && 1 == gMachineInfo.Calib )  || 1 == gMachineInfo.Manual )
			{
				if(gMachineInfo.OilAccuPressure_Extrlift < gMachineFix.OilAccu_Extrlift.AccuPressureStart)
				{
					ChargeFlag_Extrlift = 1;
				}
				else
				{
					ChargeFlag_Extrlift = 0;
				}
			}
			else if( 1 == gMachineFix.Option.bOilAccu_Extrlift_DisChar_Calib && 1 == gMachineInfo.Calib )
			{
				ChargeFlag_Extrlift = 0;
				ChargeState_Extrlift = 0;
			}
		}

		switch (ChargeState_Extrlift)
		{
			case 0:	//StandStill
				gMachineOut.Q_Charge_Extrlift	=	0;
				gMachineOut.P_Charge_Extrlift	=   0;
				gMachineOut.AccuChargeValve_Extrlift = 0;
				timeCount_Extr = 0;
				accChargeValveDelayTimeCnt_Extr = 0;
				accChargeValveTimeCount_Extr = 0;

				if(1 == ChargeFlag_Extrlift)
				{
					ChargeFlag_Extrlift = 0;
					ChargeState_Extrlift = 1;
				}
				break;

			case 1: //Charging

				accChargeValveDelayTimeCnt_Extr ++;
				if(accChargeValveDelayTimeCnt_Extr * tTask > gUserFix_new.AccChargeValve_Extrlfit_DlyTime || 1 == accChargeValveDelayDoneOnce_Extr )
				{
					accChargeValveDelayDoneOnce_Extr = 1;

					gMachineOut.AccuChargeValve_Extrlift	= 1;
					gMachineOut.Q_Charge_Extrlift			= gMachineFix.OilAccu_Extrlift.AccuFlow;
					gMachineOut.P_Charge_Extrlift			= gMachineFix.OilAccu_Extrlift.AccuChargePressure;
					timeCount_Extr ++;
					accChargeValveTimeCount_Extr ++;
					if(timeCount_Extr * tTask > gMachineFix.OilAccu_Extrlift.AccuTimeout)
					{
						//				gAlarm.AccuChargeError = 1;
					}
				}

				if(gMachineInfo.OilAccuPressure_Extrlift > gMachineFix.OilAccu_Extrlift.AccuPressureStop)
				{
					ChargeState_Extrlift = 0;
				}

				break;

		}

		RelieveCount_Extr = 15000;   /* time = 15000 * tTask this task means 300s */

	}
	else
	{
		ChargeState_Extrlift = 0;
		timeCount_Extr = 0;
		accChargeValveDelayTimeCnt_Extr = 0;
		accChargeValveDelayDoneOnce_Extr = 0;
		gMachineOut.AccuChargeValve_Extrlift  = 0;
		gMachineOut.Q_Charge_Extrlift	= 0;
		gMachineOut.P_Charge_Extrlift	= 0;
		gMachineOut.ChargeHold_Extrlift = 0;/*Reset valve*/
		if(RelieveCount_Extr > 0)RelieveCount_Extr--;

		if(1 == RelieveCount_Extr)
		{
			if(gMachineInfo.OilAccuPressure_Extrlift > 20)
			{
				/*gAlarm.AccuRelieveError = 1;*/
			}
		}
	}/* if(1 == gMachineOut.OilPump)*/

	oldChargeState_Extrlift = ChargeState_Extrlift;
	chargeTime_Extr = timeCount_Extr * tTask;
	accChargeValveDelayTime_Extr = accChargeValveDelayTimeCnt_Extr * tTask;
	accChargeValveTime_Extr = accChargeValveTimeCount_Extr * tTask;

	/* 2018.7.11 Albert High Pressure motor enable*/
	//	if(1 == gMacOption.HighPrsMotorEnable)
	//		gMachineOut.HighPrsMotorOn = gMachineOut.OilPump;
	//	else
	//		gMachineOut.HighPrsMotorOn = 0;
	gMachineOut.HighPrsMotorOn =1;

	//	gMachineOut.AccuChargeValve = gMachineIn.OilPumpRunning;

	/* ------------ 抬頭蓄壓器压力可以 ------------ */
	if(gMachineInfo.OilAccuPressure_Extrlift > gMachineFix.OilAccu_Extrlift.AccuPressureStart)
	{
		gMachineInfo.IsAccuOK_Extrlift = 1;
	}
	else
	{
		gMachineInfo.IsAccuOK_Extrlift = 0;
	}

	/* ------------------------------------------------ */

	if (1==gMacOption.OilPumpStartMode)
	{
		if ((1 == gMachineOut.OilPump) && (0==gMachineIn.OilPumpOk_DI))
		{
			OilPumpDetectTime=	tTask +OilPumpDetectTime;
			if (OilPumpDetectTime >= gUserPara.OilPumpDetectTime)
			{
				gMachineOut.OilPump=0;
				gAlarm.OilPumpErr = 1;
			}

		}
		else
		{
			OilPumpDetectTime=0;
		}
	}
	else
	{
		OilPumpDetectTime=0; //ipis0315
	}

	/* ------------ 抬頭/加壓馬達 ------------ */
	if(1 == gMacOption.HighPrsMotorEnable)
	{
		gMachineOut.HighPrsMotorOn = gMachineOut.OilPump;
	}
	else
	{
		gMachineOut.HighPrsMotorOn = 0;
	}

}/* end of _CYCLIC */
```

#### oil_accu.var
```iecst
VAR
	tTask : REAL := 0.0;
	RTInfo_Task : RTInfo := (0);
	RelieveCount : UDINT;
	timeCount : UDINT;
	chargeTime : REAL;
	ChargeState : USINT;
	ChargeFlag : USINT;
	oldChargeState : USINT;
	OilPumpDetectTime : REAL;
	OilPumpDelayTime : REAL;
	accChargeValveDelayTime : REAL;
	accChargeValveTime : REAL;
	accChargeValveDelayTimeCount : UDINT;
	accChargeValveTimeCount : UDINT;
	accChargeValveDelayDoneOnce : BOOL;
END_VAR
(*Acc Extrlift*)
VAR
	ChargeState_Extrlift : USINT;
	ChargeFlag_Extrlift : USINT;
	oldChargeState_Extrlift : USINT;
	accChargeValveDelayTime_Extr : REAL;
	accChargeValveTime_Extr : REAL;
	accChargeValveDelayTimeCnt_Extr : UDINT;
	accChargeValveTimeCount_Extr : UDINT;
	accChargeValveDelayDoneOnce_Extr : BOOL;
	timeCount_Extr : UDINT;
	RelieveCount_Extr : UDINT;
	chargeTime_Extr : REAL;
END_VAR
```

### Program Logical/machine/alarm (ANSIC, version 1.00.0) - alarm info
